LIN {X 0.032,Y -161.435,Z 1812.829,A 0.000,B 0.000,C 90.000,E1 149.282} C_DIS
LIN {X 0.039,Y -165.636,Z 1812.810,A 0.000,B 0.000,C 90.000,E1 145.754} C_DIS
LIN {X 0.022,Y -170.567,Z 1812.790,A 0.000,B 0.000,C 90.000,E1 142.271} C_DIS
LIN {X -0.071,Y -175.445,Z 1812.771,A 0.000,B 0.000,C 90.000,E1 138.852} C_DIS
LIN {X 0.045,Y -181.069,Z 1812.752,A 0.000,B 0.000,C 90.000,E1 135.405} C_DIS
LIN {X 0.036,Y -186.507,Z 1812.734,A 0.000,B 0.000,C 90.000,E1 132.043} C_DIS
LIN {X -0.021,Y -191.126,Z 1812.720,A 0.000,B 0.000,C 90.000,E1 129.564} C_DIS
LIN {X -0.101,Y -196.923,Z 1812.702,A 0.000,B 0.000,C 90.000,E1 126.297} C_DIS
LIN {X 0.093,Y -200.186,Z 1812.692,A 0.000,B 0.000,C 90.000,E1 124.612} C_DIS
LIN {X 0.089,Y -207.681,Z 1812.670,A 0.000,B 0.000,C 90.000,E1 120.590} C_DIS
LIN {X -0.010,Y -210.869,Z 1812.661,A 0.000,B 0.000,C 90.000,E1 119.027} C_DIS
LIN {X 0.101,Y -216.728,Z 1812.644,A 0.000,B 0.000,C 90.000,E1 115.848} C_DIS
LIN {X -0.080,Y -219.791,Z 1812.635,A 0.000,B 0.000,C 90.000,E1 114.335} C_DIS
LIN {X 0.010,Y -224.007,Z 1812.622,A 0.000,B 0.000,C 90.000,E1 111.897} C_DIS
LIN {X -0.023,Y -283.286,Z 1812.622,A 0.000,B 0.000,C 90.000,E1 111.897} C_DIS
LIN {X -0.096,Y -286.266,Z 1812.621,A 0.000,B 0.000,C 90.000,E1 111.844} C_DIS
LIN {X -0.059,Y -291.015,Z 1812.620,A 0.000,B 0.000,C 90.000,E1 111.535} C_DIS
LIN {X -0.019,Y -293.753,Z 1812.618,A 0.000,B 0.000,C 90.000,E1 111.227} C_DIS
LIN {X -0.009,Y -295.802,Z 1812.616,A 0.000,B 0.000,C 90.000,E1 110.918} C_DIS
LIN {X 0.132,Y -308.844,Z 1812.604,A 0.000,B 0.000,C 90.000,E1 108.598} C_DIS
LIN {X -0.084,Y -323.366,Z 1812.591,A 0.000,B 0.000,C 90.000,E1 106.370} C_DIS
LIN {X -0.136,Y -336.996,Z 1812.580,A 0.000,B 0.000,C 90.000,E1 104.481} C_DIS
LIN {X 0.084,Y -351.807,Z 1812.570,A 0.000,B 0.000,C 90.000,E1 102.591} C_DIS
LIN {X 0.058,Y -370.188,Z 1812.559,A 0.000,B 0.000,C 90.000,E1 100.546} C_DIS
LIN {X 0.090,Y -388.999,Z 1812.548,A 0.000,B 0.000,C 90.000,E1 98.681} C_DIS
LIN {X -0.052,Y -408.229,Z 1812.539,A 0.000,B 0.000,C 90.000,E1 97.004} C_DIS
LIN {X 0.143,Y -430.586,Z 1812.529,A 0.000,B 0.000,C 90.000,E1 95.220} C_DIS
LIN {X -0.141,Y -439.005,Z 1812.526,A 0.000,B 0.000,C 90.000,E1 94.645} C_DIS
LIN {X 0.070,Y -441.196,Z 1812.525,A 0.000,B 0.000,C 90.000,E1 94.416} C_DIS
LIN {X -0.017,Y -443.172,Z 1812.523,A 0.000,B 0.000,C 90.000,E1 94.188} C_DIS
LIN {X -0.073,Y -444.688,Z 1812.522,A 0.000,B 0.000,C 90.000,E1 93.955} C_DIS
LIN {X 0.104,Y -445.961,Z 1812.521,A 0.000,B 0.000,C 90.000,E1 93.669} C_DIS
LIN {X -0.162,Y -446.906,Z 1812.519,A 0.000,B 0.000,C 90.000,E1 93.440} C_DIS
LIN {X -0.206,Y -447.977,Z 1812.516,A 0.000,B 0.000,C 90.000,E1 92.922} C_DIS
LIN {X 0.178,Y -448.095,Z 1812.513,A 0.000,B 0.000,C 90.000,E1 92.350} C_DIS
LIN {X 0.126,Y -447.279,Z 1812.510,A 0.000,B 0.000,C 90.000,E1 91.835} C_DIS
LIN {X 0.086,Y -445.405,Z 1812.507,A 0.000,B 0.000,C 90.000,E1 91.318} C_DIS
LIN {X 0.029,Y -442.300,Z 1812.505,A 0.000,B 0.000,C 90.000,E1 90.802} C_DIS
LIN {X 0.055,Y -429.109,Z 1812.493,A 0.000,B 0.000,C 90.000,E1 88.682} C_DIS
LIN {X 0.115,Y -417.352,Z 1812.482,A 0.000,B 0.000,C 90.000,E1 86.788} C_DIS
LIN {X -0.123,Y -407.220,Z 1812.473,A 0.000,B 0.000,C 90.000,E1 85.179} C_DIS
LIN {X -0.062,Y -395.313,Z 1812.462,A 0.000,B 0.000,C 90.000,E1 83.223} C_DIS
LIN {X -0.160,Y -383.361,Z 1812.451,A 0.000,B 0.000,C 90.000,E1 81.254} C_DIS
LIN {X -0.061,Y -369.748,Z 1812.438,A 0.000,B 0.000,C 90.000,E1 78.926} C_DIS
LIN {X 0.062,Y -351.961,Z 1812.420,A 0.000,B 0.000,C 90.000,E1 75.644} C_DIS
LIN {X 0.049,Y -338.260,Z 1812.405,A 0.000,B 0.000,C 90.000,E1 72.906} C_DIS
LIN {X 0.047,Y -327.877,Z 1812.393,A 0.000,B 0.000,C 90.000,E1 70.732} C_DIS
LIN {X 0.147,Y -313.492,Z 1812.375,A 0.000,B 0.000,C 90.000,E1 67.539} C_DIS
LIN {X -0.191,Y -307.408,Z 1812.367,A 0.000,B 0.000,C 90.000,E1 66.177} C_DIS
LIN {X 0.160,Y -307.426,Z 1812.367,A 0.000,B 0.000,C 90.000,E1 66.102} C_DIS
LIN {X -0.061,Y -313.588,Z 1812.357,A 0.000,B 0.000,C 90.000,E1 64.332} C_DIS
LIN {X -0.097,Y -315.039,Z 1812.354,A 0.000,B 0.000,C 90.000,E1 63.691} C_DIS
LIN {X 0.156,Y -314.850,Z 1812.350,A 0.000,B 0.000,C 90.000,E1 62.999} C_DIS
LIN {X 0.136,Y -314.057,Z 1812.347,A 0.000,B 0.000,C 90.000,E1 62.359} C_DIS
LIN {X -0.163,Y -312.890,Z 1812.343,A 0.000,B 0.000,C 90.000,E1 61.769} C_DIS
LIN {X -0.040,Y -311.499,Z 1812.339,A 0.000,B 0.000,C 90.000,E1 61.101} C_DIS
LIN {X -0.077,Y -309.924,Z 1812.336,A 0.000,B 0.000,C 90.000,E1 60.461} C_DIS
LIN {X -0.029,Y -306.298,Z 1812.329,A 0.000,B 0.000,C 90.000,E1 59.154} C_DIS
LIN {X -0.131,Y -302.278,Z 1812.321,A 0.000,B 0.000,C 90.000,E1 57.867} C_DIS
LIN {X -0.082,Y -295.784,Z 1812.310,A 0.000,B 0.000,C 90.000,E1 55.881} C_DIS
LIN {X -0.007,Y -288.929,Z 1812.299,A 0.000,B 0.000,C 90.000,E1 53.863} C_DIS
LIN {X -0.008,Y -280.697,Z 1812.286,A 0.000,B 0.000,C 90.000,E1 51.492} C_DIS
LIN {X 0.037,Y -271.250,Z 1812.271,A 0.000,B 0.000,C 90.000,E1 48.728} C_DIS
LIN {X 0.001,Y -261.931,Z 1812.255,A 0.000,B 0.000,C 90.000,E1 45.931} C_DIS
LIN {X -0.082,Y -252.705,Z 1812.239,A 0.000,B 0.000,C 90.000,E1 43.095} C_DIS
LIN {X -0.014,Y -243.505,Z 1812.223,A 0.000,B 0.000,C 90.000,E1 40.172} C_DIS
LIN {X -0.137,Y -233.607,Z 1812.205,A 0.000,B 0.000,C 90.000,E1 36.870} C_DIS
LIN {X -0.042,Y -225.249,Z 1812.188,A 0.000,B 0.000,C 90.000,E1 33.833} C_DIS
LIN {X 0.033,Y -217.435,Z 1812.171,A 0.000,B 0.000,C 90.000,E1 30.747} C_DIS
LIN {X -0.006,Y -210.224,Z 1812.154,A 0.000,B 0.000,C 90.000,E1 27.641} C_DIS
LIN {X 0.043,Y -203.763,Z 1812.136,A 0.000,B 0.000,C 90.000,E1 24.463} C_DIS
LIN {X -0.047,Y -198.066,Z 1812.118,A 0.000,B 0.000,C 90.000,E1 21.280} C_DIS
LIN {X 0.062,Y -193.373,Z 1812.100,A 0.000,B 0.000,C 90.000,E1 18.000} C_DIS
LIN {X 0.064,Y -189.471,Z 1812.082,A 0.000,B 0.000,C 90.000,E1 14.717} C_DIS
LIN {X -0.020,Y -185.638,Z 1812.059,A 0.000,B 0.000,C 90.000,E1 10.602} C_DIS
LIN {X 0.045,Y -182.389,Z 1812.031,A 0.000,B 0.000,C 90.000,E1 5.568} C_DIS
LIN {X 0.015,Y -180.060,Z 1811.993,A 0.000,B 0.000,C 90.000,E1 358.682} C_DIS
LIN {X -0.031,Y -179.755,Z 1811.965,A 0.000,B 0.000,C 90.000,E1 353.628} C_DIS
LIN {X 0.009,Y -180.652,Z 1811.932,A 0.000,B 0.000,C 90.000,E1 347.701} C_DIS
LIN {X 0.001,Y -183.190,Z 1811.894,A 0.000,B 0.000,C 90.000,E1 340.967} C_DIS
LIN {X 0.075,Y -186.231,Z 1811.866,A 0.000,B 0.000,C 90.000,E1 335.921} C_DIS
LIN {X -0.051,Y -190.006,Z 1811.839,A 0.000,B 0.000,C 90.000,E1 330.973} C_DIS
LIN {X 0.006,Y -193.787,Z 1811.816,A 0.000,B 0.000,C 90.000,E1 326.834} C_DIS
LIN {X -0.044,Y -198.367,Z 1811.793,A 0.000,B 0.000,C 90.000,E1 322.763} C_DIS
LIN {X -0.102,Y -202.967,Z 1811.775,A 0.000,B 0.000,C 90.000,E1 319.542} C_DIS
LIN {X 0.000,Y -207.266,Z 1811.762,A 0.000,B 0.000,C 90.000,E1 317.106} C_DIS
LIN {X 0.102,Y -210.593,Z 1811.753,A 0.000,B 0.000,C 90.000,E1 315.486} C_DIS
LIN {X -0.006,Y -215.466,Z 1811.742,A 0.000,B 0.000,C 90.000,E1 313.542} C_DIS
LIN {X -0.087,Y -220.034,Z 1811.733,A 0.000,B 0.000,C 90.000,E1 312.000} C_DIS
LIN {X -0.108,Y -225.309,Z 1811.725,A 0.000,B 0.000,C 90.000,E1 310.458} C_DIS
LIN {X -0.036,Y -231.428,Z 1811.716,A 0.000,B 0.000,C 90.000,E1 308.910} C_DIS
LIN {X -0.060,Y -239.958,Z 1811.706,A 0.000,B 0.000,C 90.000,E1 307.030} C_DIS
LIN {X 0.061,Y -247.523,Z 1811.697,A 0.000,B 0.000,C 90.000,E1 305.518} C_DIS
LIN {X -0.111,Y -259.882,Z 1811.685,A 0.000,B 0.000,C 90.000,E1 303.372} C_DIS
LIN {X -0.111,Y -278.018,Z 1811.670,A 0.000,B 0.000,C 90.000,E1 300.541} C_DIS
LIN {X -0.137,Y -292.641,Z 1811.658,A 0.000,B 0.000,C 90.000,E1 298.487} C_DIS
LIN {X 0.030,Y -312.773,Z 1811.643,A 0.000,B 0.000,C 90.000,E1 295.796} C_DIS
LIN {X -0.102,Y -325.534,Z 1811.634,A 0.000,B 0.000,C 90.000,E1 294.207} C_DIS
LIN {X 0.124,Y -338.158,Z 1811.626,A 0.000,B 0.000,C 90.000,E1 292.589} C_DIS
LIN {X 0.124,Y -350.256,Z 1811.617,A 0.000,B 0.000,C 90.000,E1 291.046} C_DIS
LIN {X -0.127,Y -357.136,Z 1811.612,A 0.000,B 0.000,C 90.000,E1 290.174} C_DIS
LIN {X -0.100,Y -363.479,Z 1811.607,A 0.000,B 0.000,C 90.000,E1 289.268} C_DIS
LIN {X -0.016,Y -369.167,Z 1811.602,A 0.000,B 0.000,C 90.000,E1 288.362} C_DIS
LIN {X 0.133,Y -374.100,Z 1811.597,A 0.000,B 0.000,C 90.000,E1 287.457} C_DIS
LIN {X -0.141,Y -376.895,Z 1811.594,A 0.000,B 0.000,C 90.000,E1 286.913} C_DIS
LIN {X -0.035,Y -380.307,Z 1811.589,A 0.000,B 0.000,C 90.000,E1 286.024} C_DIS
LIN {X 0.093,Y -382.192,Z 1811.586,A 0.000,B 0.000,C 90.000,E1 285.426} C_DIS
LIN {X 0.227,Y -383.682,Z 1811.583,A 0.000,B 0.000,C 90.000,E1 284.828} C_DIS
LIN {X -0.099,Y -384.794,Z 1811.579,A 0.000,B 0.000,C 90.000,E1 284.300} C_DIS
LIN {X 0.053,Y -385.474,Z 1811.576,A 0.000,B 0.000,C 90.000,E1 283.703} C_DIS
LIN {X 0.119,Y -385.774,Z 1811.573,A 0.000,B 0.000,C 90.000,E1 283.119} C_DIS
LIN {X -0.184,Y -385.679,Z 1811.570,A 0.000,B 0.000,C 90.000,E1 282.591} C_DIS
LIN {X -0.109,Y -385.140,Z 1811.567,A 0.000,B 0.000,C 90.000,E1 282.007} C_DIS
LIN {X -0.032,Y -384.209,Z 1811.563,A 0.000,B 0.000,C 90.000,E1 281.422} C_DIS
LIN {X 0.040,Y -382.866,Z 1811.560,A 0.000,B 0.000,C 90.000,E1 280.838} C_DIS
LIN {X 0.106,Y -381.176,Z 1811.557,A 0.000,B 0.000,C 90.000,E1 280.254} C_DIS
LIN {X 0.183,Y -378.076,Z 1811.552,A 0.000,B 0.000,C 90.000,E1 279.378} C_DIS
LIN {X 0.168,Y -374.427,Z 1811.547,A 0.000,B 0.000,C 90.000,E1 278.511} C_DIS
LIN {X 0.118,Y -370.187,Z 1811.543,A 0.000,B 0.000,C 90.000,E1 277.644} C_DIS
LIN {X 0.037,Y -365.150,Z 1811.538,A 0.000,B 0.000,C 90.000,E1 276.777} C_DIS
LIN {X -0.093,Y -359.173,Z 1811.533,A 0.000,B 0.000,C 90.000,E1 275.910} C_DIS
LIN {X 0.136,Y -354.573,Z 1811.529,A 0.000,B 0.000,C 90.000,E1 275.277} C_DIS
LIN {X -0.016,Y -349.295,Z 1811.526,A 0.000,B 0.000,C 90.000,E1 274.702} C_DIS
LIN {X -0.063,Y -340.684,Z 1811.521,A 0.000,B 0.000,C 90.000,E1 273.841} C_DIS
LIN {X 0.124,Y -334.523,Z 1811.518,A 0.000,B 0.000,C 90.000,E1 273.269} C_DIS
LIN {X -0.040,Y -328.291,Z 1811.516,A 0.000,B 0.000,C 90.000,E1 272.808} C_DIS
LIN {X 0.015,Y -321.798,Z 1811.513,A 0.000,B 0.000,C 90.000,E1 272.350} C_DIS
LIN {X 0.017,Y -315.063,Z 1811.511,A 0.000,B 0.000,C 90.000,E1 271.949} C_DIS
LIN {X -0.002,Y -308.039,Z 1811.509,A 0.000,B 0.000,C 90.000,E1 271.604} C_DIS
LIN {X -0.036,Y -300.665,Z 1811.507,A 0.000,B 0.000,C 90.000,E1 271.318} C_DIS
LIN {X -0.024,Y -293.429,Z 1811.506,A 0.000,B 0.000,C 90.000,E1 271.088} C_DIS
LIN {X 0.084,Y -282.213,Z 1811.505,A 0.000,B 0.000,C 90.000,E1 270.802} C_DIS
LIN {X 0.083,Y -267.546,Z 1811.503,A 0.000,B 0.000,C 90.000,E1 270.516} C_DIS
LIN {X -0.067,Y -252.024,Z 1811.501,A 0.000,B 0.000,C 90.000,E1 270.286} C_DIS
LIN {X -0.055,Y -241.026,Z 1811.501,A 0.000,B 0.000,C 90.000,E1 270.172} C_DIS
LIN {X 0.028,Y -234.816,Z 1811.501,A 0.000,B 0.000,C 90.000,E1 270.115} C_DIS
LIN {X -0.002,Y -181.574,Z 1811.501,A 0.000,B 0.000,C 90.000,E1 270.115} C_DIS
LIN {X 0.084,Y -180.908,Z 1811.475,A 0.000,B 0.000,C 90.000,E1 265.527} C_DIS
LIN {X -0.038,Y -180.772,Z 1811.471,A 0.000,B 0.000,C 90.000,E1 264.723} C_DIS
LIN {X 0.033,Y -178.867,Z 1811.443,A 0.000,B 0.000,C 90.000,E1 259.634} C_DIS
LIN {X -0.066,Y -175.910,Z 1811.414,A 0.000,B 0.000,C 90.000,E1 254.574} C_DIS
LIN {X -0.010,Y -174.597,Z 1811.405,A 0.000,B 0.000,C 90.000,E1 252.851} C_DIS
LIN {X -0.083,Y -171.579,Z 1811.381,A 0.000,B 0.000,C 90.000,E1 248.592} C_DIS
LIN {X -0.093,Y -167.802,Z 1811.357,A 0.000,B 0.000,C 90.000,E1 244.280} C_DIS
LIN {X 0.072,Y -166.520,Z 1811.347,A 0.000,B 0.000,C 90.000,E1 242.487} C_DIS
LIN {X 0.060,Y -162.521,Z 1811.323,A 0.000,B 0.000,C 90.000,E1 238.122} C_DIS
LIN {X 0.031,Y -161.194,Z 1811.313,A 0.000,B 0.000,C 90.000,E1 236.373} C_DIS
LIN {X -0.066,Y -157.205,Z 1811.289,A 0.000,B 0.000,C 90.000,E1 231.984} C_DIS
LIN {X -0.043,Y -155.933,Z 1811.279,A 0.000,B 0.000,C 90.000,E1 230.194} C_DIS
LIN {X -0.083,Y -152.185,Z 1811.254,A 0.000,B 0.000,C 90.000,E1 225.729} C_DIS
LIN {X -0.062,Y -150.432,Z 1811.239,A 0.000,B 0.000,C 90.000,E1 223.014} C_DIS
LIN {X -0.033,Y -147.159,Z 1811.214,A 0.000,B 0.000,C 90.000,E1 218.463} C_DIS
LIN {X -0.067,Y -145.174,Z 1811.193,A 0.000,B 0.000,C 90.000,E1 214.818} C_DIS
LIN {X -0.031,Y -142.322,Z 1811.163,A 0.000,B 0.000,C 90.000,E1 209.283} C_DIS
LIN {X -0.037,Y -141.712,Z 1811.152,A 0.000,B 0.000,C 90.000,E1 207.436} C_DIS
LIN {X 0.012,Y -139.473,Z 1811.116,A 0.000,B 0.000,C 90.000,E1 200.918} C_DIS
LIN {X -0.067,Y -139.204,Z 1811.106,A 0.000,B 0.000,C 90.000,E1 199.087} C_DIS
LIN {X -0.008,Y -138.329,Z 1811.054,A 0.000,B 0.000,C 90.000,E1 189.726} C_DIS
LIN {X -0.005,Y -139.439,Z 1811.007,A 0.000,B 0.000,C 90.000,E1 181.318} C_DIS
LIN {X -0.066,Y -140.971,Z 1810.976,A 0.000,B 0.000,C 90.000,E1 175.755} C_DIS
LIN {X 0.025,Y -142.727,Z 1810.956,A 0.000,B 0.000,C 90.000,E1 172.008} C_DIS
LIN {X -0.017,Y -145.111,Z 1810.930,A 0.000,B 0.000,C 90.000,E1 167.409} C_DIS
LIN {X -0.022,Y -147.735,Z 1810.910,A 0.000,B 0.000,C 90.000,E1 163.740} C_DIS
LIN {X 0.059,Y -150.398,Z 1810.889,A 0.000,B 0.000,C 90.000,E1 160.061} C_DIS
LIN {X -0.066,Y -153.834,Z 1810.869,A 0.000,B 0.000,C 90.000,E1 156.485} C_DIS
LIN {X -0.007,Y -157.244,Z 1810.849,A 0.000,B 0.000,C 90.000,E1 152.871} C_DIS
LIN {X -0.067,Y -161.416,Z 1810.829,A 0.000,B 0.000,C 90.000,E1 149.331} C_DIS
LIN {X -0.057,Y -165.617,Z 1810.810,A 0.000,B 0.000,C 90.000,E1 145.801} C_DIS
LIN {X 0.063,Y -170.546,Z 1810.791,A 0.000,B 0.000,C 90.000,E1 142.271} C_DIS
LIN {X -0.029,Y -175.424,Z 1810.771,A 0.000,B 0.000,C 90.000,E1 138.852} C_DIS
LIN {X 0.088,Y -181.048,Z 1810.752,A 0.000,B 0.000,C 90.000,E1 135.405} C_DIS
LIN {X -0.046,Y -186.483,Z 1810.734,A 0.000,B 0.000,C 90.000,E1 132.081} C_DIS
LIN {X 0.022,Y -191.105,Z 1810.720,A 0.000,B 0.000,C 90.000,E1 129.564} C_DIS
LIN {X -0.057,Y -196.898,Z 1810.702,A 0.000,B 0.000,C 90.000,E1 126.297} C_DIS
LIN {X -0.026,Y -200.159,Z 1810.693,A 0.000,B 0.000,C 90.000,E1 124.659} C_DIS
LIN {X 0.030,Y -207.655,Z 1810.670,A 0.000,B 0.000,C 90.000,E1 120.620} C_DIS
LIN {X 0.037,Y -210.848,Z 1810.661,A 0.000,B 0.000,C 90.000,E1 119.027} C_DIS
LIN {X -0.047,Y -216.703,Z 1810.644,A 0.000,B 0.000,C 90.000,E1 115.899} C_DIS
LIN {X -0.033,Y -219.771,Z 1810.635,A 0.000,B 0.000,C 90.000,E1 114.335} C_DIS
LIN {X 0.002,Y -224.010,Z 1810.622,A 0.000,B 0.000,C 90.000,E1 111.897} C_DIS
LIN {X -0.033,Y -283.663,Z 1810.622,A 0.000,B 0.000,C 90.000,E1 111.897} C_DIS
LIN {X -0.036,Y -285.968,Z 1810.621,A 0.000,B 0.000,C 90.000,E1 111.844} C_DIS
LIN {X 0.003,Y -290.889,Z 1810.620,A 0.000,B 0.000,C 90.000,E1 111.535} C_DIS
LIN {X 0.044,Y -293.661,Z 1810.618,A 0.000,B 0.000,C 90.000,E1 111.227} C_DIS
LIN {X 0.069,Y -295.712,Z 1810.616,A 0.000,B 0.000,C 90.000,E1 110.918} C_DIS
LIN {X -0.065,Y -308.735,Z 1810.604,A 0.000,B 0.000,C 90.000,E1 108.652} C_DIS
LIN {X -0.076,Y -323.246,Z 1810.591,A 0.000,B 0.000,C 90.000,E1 106.386} C_DIS
LIN {X -0.037,Y -336.866,Z 1810.580,A 0.000,B 0.000,C 90.000,E1 104.481} C_DIS
LIN {X -0.158,Y -351.666,Z 1810.570,A 0.000,B 0.000,C 90.000,E1 102.647} C_DIS
LIN {X 0.155,Y -370.043,Z 1810.559,A 0.000,B 0.000,C 90.000,E1 100.546} C_DIS
LIN {X 0.125,Y -388.849,Z 1810.548,A 0.000,B 0.000,C 90.000,E1 98.690} C_DIS
LIN {X 0.037,Y -408.077,Z 1810.539,A 0.000,B 0.000,C 90.000,E1 97.004} C_DIS
LIN {X -0.200,Y -430.431,Z 1810.529,A 0.000,B 0.000,C 90.000,E1 95.277} C_DIS
LIN {X -0.057,Y -438.863,Z 1810.526,A 0.000,B 0.000,C 90.000,E1 94.645} C_DIS
LIN {X 0.153,Y -441.087,Z 1810.525,A 0.000,B 0.000,C 90.000,E1 94.416} C_DIS
LIN {X 0.084,Y -443.070,Z 1810.523,A 0.000,B 0.000,C 90.000,E1 94.188} C_DIS
LIN {X 0.047,Y -444.593,Z 1810.522,A 0.000,B 0.000,C 90.000,E1 93.955} C_DIS
LIN {X 0.224,Y -445.885,Z 1810.521,A 0.000,B 0.000,C 90.000,E1 93.669} C_DIS
LIN {X -0.042,Y -446.847,Z 1810.519,A 0.000,B 0.000,C 90.000,E1 93.440} C_DIS
LIN {X -0.087,Y -447.947,Z 1810.516,A 0.000,B 0.000,C 90.000,E1 92.922} C_DIS
LIN {X -0.150,Y -448.091,Z 1810.513,A 0.000,B 0.000,C 90.000,E1 92.407} C_DIS
LIN {X -0.203,Y -447.302,Z 1810.510,A 0.000,B 0.000,C 90.000,E1 91.892} C_DIS
LIN {X 0.204,Y -445.459,Z 1810.507,A 0.000,B 0.000,C 90.000,E1 91.318} C_DIS
LIN {X 0.147,Y -442.378,Z 1810.505,A 0.000,B 0.000,C 90.000,E1 90.802} C_DIS
LIN {X 0.172,Y -429.186,Z 1810.493,A 0.000,B 0.000,C 90.000,E1 88.682} C_DIS
LIN {X -0.187,Y -417.432,Z 1810.482,A 0.000,B 0.000,C 90.000,E1 86.846} C_DIS
LIN {X -0.010,Y -407.300,Z 1810.473,A 0.000,B 0.000,C 90.000,E1 85.179} C_DIS
LIN {X 0.050,Y -395.395,Z 1810.462,A 0.000,B 0.000,C 90.000,E1 83.223} C_DIS
LIN {X -0.050,Y -383.442,Z 1810.451,A 0.000,B 0.000,C 90.000,E1 81.254} C_DIS
LIN {X 0.047,Y -369.825,Z 1810.438,A 0.000,B 0.000,C 90.000,E1 78.926} C_DIS
LIN {X -0.174,Y -352.031,Z 1810.420,A 0.000,B 0.000,C 90.000,E1 75.700} C_DIS
LIN {X 0.152,Y -338.326,Z 1810.405,A 0.000,B 0.000,C 90.000,E1 72.906} C_DIS
LIN {X 0.148,Y -327.941,Z 1810.393,A 0.000,B 0.000,C 90.000,E1 70.732} C_DIS
LIN {X -0.098,Y -314.945,Z 1810.377,A 0.000,B 0.000,C 90.000,E1 67.922} C_DIS
LIN {X -0.035,Y -314.938,Z 1810.377,A 0.000,B 0.000,C 90.000,E1 67.901} C_DIS
LIN {X -0.040,Y -320.081,Z 1810.368,A 0.000,B 0.000,C 90.000,E1 66.305} C_DIS
LIN {X -0.040,Y -322.043,Z 1810.365,A 0.000,B 0.000,C 90.000,E1 65.665} C_DIS
LIN {X -0.029,Y -322.287,Z 1810.361,A 0.000,B 0.000,C 90.000,E1 65.025} C_DIS
LIN {X -0.143,Y -321.735,Z 1810.358,A 0.000,B 0.000,C 90.000,E1 64.409} C_DIS
LIN {X -0.119,Y -320.798,Z 1810.354,A 0.000,B 0.000,C 90.000,E1 63.768} C_DIS
LIN {X -0.097,Y -319.593,Z 1810.351,A 0.000,B 0.000,C 90.000,E1 63.127} C_DIS
LIN {X -0.074,Y -316.589,Z 1810.344,A 0.000,B 0.000,C 90.000,E1 61.847} C_DIS
LIN {X 0.058,Y -313.018,Z 1810.336,A 0.000,B 0.000,C 90.000,E1 60.539} C_DIS
LIN {X 0.034,Y -308.980,Z 1810.329,A 0.000,B 0.000,C 90.000,E1 59.253} C_DIS
LIN {X -0.151,Y -303.508,Z 1810.320,A 0.000,B 0.000,C 90.000,E1 57.661} C_DIS
LIN {X -0.095,Y -296.538,Z 1810.309,A 0.000,B 0.000,C 90.000,E1 55.674} C_DIS
LIN {X 0.157,Y -289.302,Z 1810.298,A 0.000,B 0.000,C 90.000,E1 53.623} C_DIS
LIN {X -0.053,Y -280.703,Z 1810.285,A 0.000,B 0.000,C 90.000,E1 51.295} C_DIS
LIN {X 0.006,Y -270.889,Z 1810.270,A 0.000,B 0.000,C 90.000,E1 48.528} C_DIS
LIN {X -0.031,Y -261.234,Z 1810.254,A 0.000,B 0.000,C 90.000,E1 45.729} C_DIS
LIN {X 0.049,Y -251.694,Z 1810.238,A 0.000,B 0.000,C 90.000,E1 42.852} C_DIS
LIN {X 0.076,Y -241.310,Z 1810.220,A 0.000,B 0.000,C 90.000,E1 39.564} C_DIS
LIN {X -0.047,Y -233.632,Z 1810.205,A 0.000,B 0.000,C 90.000,E1 36.996} C_DIS
LIN {X -0.085,Y -225.238,Z 1810.189,A 0.000,B 0.000,C 90.000,E1 33.992} C_DIS
LIN {X -0.077,Y -217.413,Z 1810.172,A 0.000,B 0.000,C 90.000,E1 30.924} C_DIS
LIN {X 0.066,Y -210.161,Z 1810.154,A 0.000,B 0.000,C 90.000,E1 27.769} C_DIS
LIN {X -0.074,Y -203.660,Z 1810.137,A 0.000,B 0.000,C 90.000,E1 24.643} C_DIS
LIN {X 0.019,Y -197.902,Z 1810.119,A 0.000,B 0.000,C 90.000,E1 21.408} C_DIS
LIN {X -0.059,Y -193.137,Z 1810.101,A 0.000,B 0.000,C 90.000,E1 18.181} C_DIS
LIN {X -0.059,Y -189.201,Z 1810.083,A 0.000,B 0.000,C 90.000,E1 14.898} C_DIS
LIN {X 0.037,Y -185.326,Z 1810.060,A 0.000,B 0.000,C 90.000,E1 10.725} C_DIS
LIN {X -0.062,Y -182.055,Z 1810.032,A 0.000,B 0.000,C 90.000,E1 5.739} C_DIS
LIN {X 0.013,Y -179.684,Z 1809.993,A 0.000,B 0.000,C 90.000,E1 358.682} C_DIS
LIN {X 0.018,Y -179.407,Z 1809.960,A 0.000,B 0.000,C 90.000,E1 352.761} C_DIS
LIN {X -0.022,Y -180.306,Z 1809.932,A 0.000,B 0.000,C 90.000,E1 347.701} C_DIS
LIN {X -0.050,Y -182.858,Z 1809.894,A 0.000,B 0.000,C 90.000,E1 340.967} C_DIS
LIN {X 0.011,Y -185.925,Z 1809.866,A 0.000,B 0.000,C 90.000,E1 335.921} C_DIS
LIN {X 0.039,Y -189.748,Z 1809.839,A 0.000,B 0.000,C 90.000,E1 330.923} C_DIS
LIN {X -0.080,Y -193.551,Z 1809.816,A 0.000,B 0.000,C 90.000,E1 326.834} C_DIS
LIN {X 0.019,Y -198.199,Z 1809.793,A 0.000,B 0.000,C 90.000,E1 322.718} C_DIS
LIN {X 0.084,Y -202.896,Z 1809.775,A 0.000,B 0.000,C 90.000,E1 319.461} C_DIS
LIN {X 0.039,Y -207.280,Z 1809.762,A 0.000,B 0.000,C 90.000,E1 317.067} C_DIS
LIN {X -0.003,Y -210.662,Z 1809.753,A 0.000,B 0.000,C 90.000,E1 315.486} C_DIS
LIN {X -0.109,Y -215.578,Z 1809.742,A 0.000,B 0.000,C 90.000,E1 313.542} C_DIS
LIN {X 0.124,Y -220.192,Z 1809.733,A 0.000,B 0.000,C 90.000,E1 311.919} C_DIS
LIN {X -0.038,Y -225.510,Z 1809.724,A 0.000,B 0.000,C 90.000,E1 310.415} C_DIS
LIN {X 0.007,Y -231.660,Z 1809.716,A 0.000,B 0.000,C 90.000,E1 308.874} C_DIS
LIN {X -0.017,Y -240.225,Z 1809.706,A 0.000,B 0.000,C 90.000,E1 306.996} C_DIS
LIN {X -0.043,Y -249.816,Z 1809.695,A 0.000,B 0.000,C 90.000,E1 305.152} C_DIS
LIN {X -0.071,Y -264.598,Z 1809.681,A 0.000,B 0.000,C 90.000,E1 302.625} C_DIS
LIN {X 0.059,Y -283.268,Z 1809.666,A 0.000,B 0.000,C 90.000,E1 299.795} C_DIS
LIN {X -0.003,Y -298.015,Z 1809.654,A 0.000,B 0.000,C 90.000,E1 297.769} C_DIS
LIN {X -0.015,Y -315.826,Z 1809.641,A 0.000,B 0.000,C 90.000,E1 295.463} C_DIS
LIN {X 0.186,Y -328.618,Z 1809.633,A 0.000,B 0.000,C 90.000,E1 293.823} C_DIS
LIN {X 0.052,Y -338.702,Z 1809.625,A 0.000,B 0.000,C 90.000,E1 292.589} C_DIS
LIN {X 0.058,Y -350.836,Z 1809.617,A 0.000,B 0.000,C 90.000,E1 291.046} C_DIS
LIN {X 0.146,Y -357.744,Z 1809.612,A 0.000,B 0.000,C 90.000,E1 290.120} C_DIS
LIN {X -0.158,Y -364.058,Z 1809.607,A 0.000,B 0.000,C 90.000,E1 289.268} C_DIS
LIN {X -0.068,Y -369.763,Z 1809.602,A 0.000,B 0.000,C 90.000,E1 288.362} C_DIS
LIN {X -0.012,Y -373.159,Z 1809.599,A 0.000,B 0.000,C 90.000,E1 287.764} C_DIS
LIN {X 0.174,Y -377.459,Z 1809.594,A 0.000,B 0.000,C 90.000,E1 286.858} C_DIS
LIN {X -0.076,Y -380.864,Z 1809.589,A 0.000,B 0.000,C 90.000,E1 286.024} C_DIS
LIN {X 0.056,Y -382.720,Z 1809.586,A 0.000,B 0.000,C 90.000,E1 285.426} C_DIS
LIN {X 0.193,Y -384.185,Z 1809.583,A 0.000,B 0.000,C 90.000,E1 284.828} C_DIS
LIN {X -0.129,Y -385.230,Z 1809.579,A 0.000,B 0.000,C 90.000,E1 284.300} C_DIS
LIN {X 0.026,Y -385.956,Z 1809.576,A 0.000,B 0.000,C 90.000,E1 283.703} C_DIS
LIN {X 0.095,Y -386.250,Z 1809.573,A 0.000,B 0.000,C 90.000,E1 283.119} C_DIS
LIN {X 0.171,Y -386.154,Z 1809.570,A 0.000,B 0.000,C 90.000,E1 282.535} C_DIS
LIN {X -0.127,Y -385.589,Z 1809.567,A 0.000,B 0.000,C 90.000,E1 282.007} C_DIS
LIN {X -0.049,Y -384.670,Z 1809.563,A 0.000,B 0.000,C 90.000,E1 281.422} C_DIS
LIN {X 0.026,Y -383.357,Z 1809.560,A 0.000,B 0.000,C 90.000,E1 280.838} C_DIS
LIN {X 0.095,Y -381.670,Z 1809.557,A 0.000,B 0.000,C 90.000,E1 280.254} C_DIS
LIN {X 0.154,Y -379.748,Z 1809.554,A 0.000,B 0.000,C 90.000,E1 279.670} C_DIS
LIN {X 0.154,Y -376.213,Z 1809.549,A 0.000,B 0.000,C 90.000,E1 278.803} C_DIS
LIN {X 0.125,Y -372.175,Z 1809.544,A 0.000,B 0.000,C 90.000,E1 277.936} C_DIS
LIN {X 0.058,Y -367.390,Z 1809.539,A 0.000,B 0.000,C 90.000,E1 277.068} C_DIS
LIN {X 0.020,Y -363.730,Z 1809.536,A 0.000,B 0.000,C 90.000,E1 276.486} C_DIS
LIN {X -0.154,Y -357.285,Z 1809.531,A 0.000,B 0.000,C 90.000,E1 275.625} C_DIS
LIN {X 0.067,Y -352.348,Z 1809.528,A 0.000,B 0.000,C 90.000,E1 274.992} C_DIS
LIN {X -0.090,Y -346.752,Z 1809.524,A 0.000,B 0.000,C 90.000,E1 274.416} C_DIS
LIN {X -0.020,Y -341.011,Z 1809.521,A 0.000,B 0.000,C 90.000,E1 273.841} C_DIS
LIN {X -0.125,Y -334.919,Z 1809.518,A 0.000,B 0.000,C 90.000,E1 273.326} C_DIS
LIN {X 0.059,Y -328.746,Z 1809.516,A 0.000,B 0.000,C 90.000,E1 272.808} C_DIS
LIN {X 0.100,Y -322.215,Z 1809.513,A 0.000,B 0.000,C 90.000,E1 272.350} C_DIS
LIN {X 0.104,Y -315.524,Z 1809.511,A 0.000,B 0.000,C 90.000,E1 271.949} C_DIS
LIN {X 0.069,Y -308.453,Z 1809.509,A 0.000,B 0.000,C 90.000,E1 271.604} C_DIS
LIN {X 0.003,Y -300.959,Z 1809.507,A 0.000,B 0.000,C 90.000,E1 271.318} C_DIS
LIN {X 0.009,Y -293.694,Z 1809.506,A 0.000,B 0.000,C 90.000,E1 271.088} C_DIS
LIN {X 0.012,Y -278.792,Z 1809.504,A 0.000,B 0.000,C 90.000,E1 270.745} C_DIS
LIN {X 0.003,Y -260.019,Z 1809.502,A 0.000,B 0.000,C 90.000,E1 270.401} C_DIS
LIN {X -0.049,Y -251.634,Z 1809.502,A 0.000,B 0.000,C 90.000,E1 270.286} C_DIS
LIN {X 0.096,Y -236.258,Z 1809.501,A 0.000,B 0.000,C 90.000,E1 270.115} C_DIS
LIN {X 0.066,Y -234.027,Z 1809.501,A 0.000,B 0.000,C 90.000,E1 270.115} C_DIS
LIN {X 0.028,Y -181.575,Z 1809.501,A 0.000,B 0.000,C 90.000,E1 270.115} C_DIS
LIN {X -0.065,Y -180.908,Z 1809.475,A 0.000,B 0.000,C 90.000,E1 265.584} C_DIS
LIN {X -0.008,Y -180.776,Z 1809.471,A 0.000,B 0.000,C 90.000,E1 264.723} C_DIS
LIN {X 0.063,Y -178.871,Z 1809.443,A 0.000,B 0.000,C 90.000,E1 259.634} C_DIS
LIN {X -0.035,Y -175.914,Z 1809.414,A 0.000,B 0.000,C 90.000,E1 254.574} C_DIS
LIN {X 0.021,Y -174.605,Z 1809.405,A 0.000,B 0.000,C 90.000,E1 252.851} C_DIS
LIN {X -0.053,Y -171.587,Z 1809.381,A 0.000,B 0.000,C 90.000,E1 248.592} C_DIS
LIN {X -0.064,Y -167.810,Z 1809.357,A 0.000,B 0.000,C 90.000,E1 244.280} C_DIS
LIN {X -0.047,Y -166.530,Z 1809.347,A 0.000,B 0.000,C 90.000,E1 242.538} C_DIS
LIN {X 0.090,Y -162.529,Z 1809.323,A 0.000,B 0.000,C 90.000,E1 238.122} C_DIS
LIN {X -0.074,Y -161.204,Z 1809.313,A 0.000,B 0.000,C 90.000,E1 236.421} C_DIS
LIN {X -0.038,Y -157.213,Z 1809.289,A 0.000,B 0.000,C 90.000,E1 231.984} C_DIS
LIN {X -0.015,Y -155.940,Z 1809.279,A 0.000,B 0.000,C 90.000,E1 230.194} C_DIS
LIN {X -0.055,Y -152.192,Z 1809.254,A 0.000,B 0.000,C 90.000,E1 225.729} C_DIS
LIN {X -0.034,Y -150.439,Z 1809.239,A 0.000,B 0.000,C 90.000,E1 223.014} C_DIS
LIN {X -0.006,Y -147.165,Z 1809.214,A 0.000,B 0.000,C 90.000,E1 218.463} C_DIS
LIN {X -0.040,Y -145.180,Z 1809.193,A 0.000,B 0.000,C 90.000,E1 214.818} C_DIS
LIN {X -0.005,Y -142.327,Z 1809.163,A 0.000,B 0.000,C 90.000,E1 209.283} C_DIS
LIN {X -0.009,Y -141.716,Z 1809.152,A 0.000,B 0.000,C 90.000,E1 207.436} C_DIS
LIN {X 0.038,Y -139.474,Z 1809.116,A 0.000,B 0.000,C 90.000,E1 200.918} C_DIS
LIN {X 0.029,Y -138.971,Z 1809.101,A 0.000,B 0.000,C 90.000,E1 198.127} C_DIS
LIN {X 0.018,Y -138.330,Z 1809.054,A 0.000,B 0.000,C 90.000,E1 189.726} C_DIS
LIN {X 0.021,Y -139.436,Z 1809.007,A 0.000,B 0.000,C 90.000,E1 181.318} C_DIS
LIN {X -0.039,Y -140.967,Z 1808.976,A 0.000,B 0.000,C 90.000,E1 175.755} C_DIS
LIN {X 0.052,Y -142.722,Z 1808.956,A 0.000,B 0.000,C 90.000,E1 172.008} C_DIS
LIN {X 0.010,Y -145.104,Z 1808.930,A 0.000,B 0.000,C 90.000,E1 167.409} C_DIS
LIN {X 0.005,Y -147.729,Z 1808.910,A 0.000,B 0.000,C 90.000,E1 163.740} C_DIS
LIN {X -0.054,Y -150.389,Z 1808.889,A 0.000,B 0.000,C 90.000,E1 160.115} C_DIS
LIN {X -0.038,Y -153.823,Z 1808.869,A 0.000,B 0.000,C 90.000,E1 156.485} C_DIS
LIN {X 0.021,Y -157.233,Z 1808.849,A 0.000,B 0.000,C 90.000,E1 152.871} C_DIS
LIN {X -0.038,Y -161.403,Z 1808.830,A 0.000,B 0.000,C 90.000,E1 149.331} C_DIS
LIN {X -0.028,Y -165.605,Z 1808.810,A 0.000,B 0.000,C 90.000,E1 145.801} C_DIS
LIN {X 0.093,Y -170.530,Z 1808.791,A 0.000,B 0.000,C 90.000,E1 142.271} C_DIS
LIN {X 0.001,Y -175.409,Z 1808.771,A 0.000,B 0.000,C 90.000,E1 138.852} C_DIS
LIN {X -0.009,Y -181.033,Z 1808.752,A 0.000,B 0.000,C 90.000,E1 135.445} C_DIS
LIN {X -0.014,Y -186.466,Z 1808.734,A 0.000,B 0.000,C 90.000,E1 132.081} C_DIS
LIN {X 0.054,Y -191.089,Z 1808.720,A 0.000,B 0.000,C 90.000,E1 129.564} C_DIS
LIN {X -0.025,Y -196.880,Z 1808.702,A 0.000,B 0.000,C 90.000,E1 126.297} C_DIS
LIN {X 0.007,Y -200.139,Z 1808.693,A 0.000,B 0.000,C 90.000,E1 124.659} C_DIS
LIN {X -0.116,Y -207.636,Z 1808.670,A 0.000,B 0.000,C 90.000,E1 120.669} C_DIS
LIN {X -0.114,Y -210.831,Z 1808.661,A 0.000,B 0.000,C 90.000,E1 119.077} C_DIS
LIN {X -0.013,Y -216.685,Z 1808.644,A 0.000,B 0.000,C 90.000,E1 115.899} C_DIS
LIN {X 0.003,Y -219.756,Z 1808.635,A 0.000,B 0.000,C 90.000,E1 114.335} C_DIS
LIN {X -0.035,Y -221.985,Z 1808.628,A 0.000,B 0.000,C 90.000,E1 113.025} C_DIS
LIN {X -0.081,Y -293.410,Z 1808.628,A 0.000,B 0.000,C 90.000,E1 113.025} C_DIS
LIN {X -0.036,Y -294.839,Z 1808.628,A 0.000,B 0.000,C 90.000,E1 113.003} C_DIS
LIN {X 0.082,Y -299.077,Z 1808.627,A 0.000,B 0.000,C 90.000,E1 112.770} C_DIS
LIN {X 0.086,Y -300.273,Z 1808.625,A 0.000,B 0.000,C 90.000,E1 112.461} C_DIS
LIN {X -0.153,Y -299.587,Z 1808.621,A 0.000,B 0.000,C 90.000,E1 111.844} C_DIS
LIN {X 0.092,Y -297.703,Z 1808.614,A 0.000,B 0.000,C 90.000,E1 110.556} C_DIS
LIN {X 0.039,Y -297.729,Z 1808.614,A 0.000,B 0.000,C 90.000,E1 110.556} C_DIS
LIN {X 0.100,Y -309.533,Z 1808.603,A 0.000,B 0.000,C 90.000,E1 108.489} C_DIS
LIN {X -0.093,Y -324.127,Z 1808.590,A 0.000,B 0.000,C 90.000,E1 106.260} C_DIS
LIN {X -0.042,Y -337.823,Z 1808.580,A 0.000,B 0.000,C 90.000,E1 104.356} C_DIS
LIN {X 0.116,Y -352.706,Z 1808.569,A 0.000,B 0.000,C 90.000,E1 102.479} C_DIS
LIN {X 0.155,Y -371.120,Z 1808.558,A 0.000,B 0.000,C 90.000,E1 100.433} C_DIS
LIN {X -0.128,Y -389.949,Z 1808.548,A 0.000,B 0.000,C 90.000,E1 98.624} C_DIS
LIN {X 0.183,Y -409.195,Z 1808.538,A 0.000,B 0.000,C 90.000,E1 96.891} C_DIS
LIN {X 0.024,Y -431.569,Z 1808.529,A 0.000,B 0.000,C 90.000,E1 95.163} C_DIS
LIN {X -0.020,Y -437.223,Z 1808.526,A 0.000,B 0.000,C 90.000,E1 94.759} C_DIS
LIN {X -0.024,Y -441.813,Z 1808.524,A 0.000,B 0.000,C 90.000,E1 94.359} C_DIS
LIN {X -0.044,Y -444.957,Z 1808.522,A 0.000,B 0.000,C 90.000,E1 93.898} C_DIS
LIN {X 0.131,Y -446.159,Z 1808.520,A 0.000,B 0.000,C 90.000,E1 93.612} C_DIS
LIN {X -0.140,Y -447.042,Z 1808.519,A 0.000,B 0.000,C 90.000,E1 93.383} C_DIS
LIN {X -0.183,Y -448.007,Z 1808.516,A 0.000,B 0.000,C 90.000,E1 92.865} C_DIS
LIN {X 0.204,Y -448.027,Z 1808.513,A 0.000,B 0.000,C 90.000,E1 92.293} C_DIS
LIN {X 0.164,Y -447.108,Z 1808.510,A 0.000,B 0.000,C 90.000,E1 91.776} C_DIS
LIN {X 0.110,Y -445.103,Z 1808.507,A 0.000,B 0.000,C 90.000,E1 91.260} C_DIS
LIN {X -0.023,Y -438.606,Z 1808.501,A 0.000,B 0.000,C 90.000,E1 90.229} C_DIS
LIN {X 0.207,Y -427.065,Z 1808.491,A 0.000,B 0.000,C 90.000,E1 88.339} C_DIS
LIN {X -0.191,Y -415.294,Z 1808.480,A 0.000,B 0.000,C 90.000,E1 86.502} C_DIS
LIN {X 0.036,Y -403.433,Z 1808.470,A 0.000,B 0.000,C 90.000,E1 84.546} C_DIS
LIN {X -0.007,Y -393.207,Z 1808.460,A 0.000,B 0.000,C 90.000,E1 82.875} C_DIS
LIN {X -0.141,Y -381.262,Z 1808.449,A 0.000,B 0.000,C 90.000,E1 80.905} C_DIS
LIN {X -0.106,Y -366.042,Z 1808.435,A 0.000,B 0.000,C 90.000,E1 78.285} C_DIS
LIN {X -0.023,Y -348.503,Z 1808.417,A 0.000,B 0.000,C 90.000,E1 74.991} C_DIS
LIN {X -0.014,Y -336.416,Z 1808.403,A 0.000,B 0.000,C 90.000,E1 72.543} C_DIS
LIN {X -0.091,Y -324.598,Z 1808.389,A 0.000,B 0.000,C 90.000,E1 70.061} C_DIS
LIN {X 0.028,Y -322.668,Z 1808.387,A 0.000,B 0.000,C 90.000,E1 69.625} C_DIS
LIN {X -0.027,Y -322.630,Z 1808.387,A 0.000,B 0.000,C 90.000,E1 69.625} C_DIS
LIN {X 0.134,Y -329.133,Z 1808.375,A 0.000,B 0.000,C 90.000,E1 67.486} C_DIS
LIN {X 0.053,Y -329.566,Z 1808.372,A 0.000,B 0.000,C 90.000,E1 66.869} C_DIS
LIN {X 0.115,Y -329.090,Z 1808.368,A 0.000,B 0.000,C 90.000,E1 66.230} C_DIS
LIN {X 0.049,Y -328.211,Z 1808.365,A 0.000,B 0.000,C 90.000,E1 65.613} C_DIS
LIN {X 0.114,Y -327.081,Z 1808.361,A 0.000,B 0.000,C 90.000,E1 64.973} C_DIS
LIN {X 0.088,Y -324.319,Z 1808.354,A 0.000,B 0.000,C 90.000,E1 63.717} C_DIS
LIN {X -0.117,Y -321.031,Z 1808.347,A 0.000,B 0.000,C 90.000,E1 62.487} C_DIS
LIN {X 0.076,Y -317.250,Z 1808.340,A 0.000,B 0.000,C 90.000,E1 61.179} C_DIS
LIN {X 0.015,Y -312.014,Z 1808.331,A 0.000,B 0.000,C 90.000,E1 59.587} C_DIS
LIN {X -0.134,Y -306.261,Z 1808.322,A 0.000,B 0.000,C 90.000,E1 57.995} C_DIS
LIN {X -0.030,Y -298.955,Z 1808.311,A 0.000,B 0.000,C 90.000,E1 56.008} C_DIS
LIN {X 0.098,Y -291.476,Z 1808.300,A 0.000,B 0.000,C 90.000,E1 53.989} C_DIS
LIN {X -0.071,Y -282.552,Z 1808.287,A 0.000,B 0.000,C 90.000,E1 51.662} C_DIS
LIN {X -0.147,Y -272.344,Z 1808.272,A 0.000,B 0.000,C 90.000,E1 48.933} C_DIS
LIN {X -0.148,Y -262.297,Z 1808.256,A 0.000,B 0.000,C 90.000,E1 46.134} C_DIS
LIN {X -0.025,Y -251.404,Z 1808.238,A 0.000,B 0.000,C 90.000,E1 42.894} C_DIS
LIN {X 0.019,Y -241.003,Z 1808.220,A 0.000,B 0.000,C 90.000,E1 39.600} C_DIS
LIN {X 0.033,Y -233.298,Z 1808.206,A 0.000,B 0.000,C 90.000,E1 36.996} C_DIS
LIN {X -0.015,Y -224.897,Z 1808.189,A 0.000,B 0.000,C 90.000,E1 33.992} C_DIS
LIN {X -0.018,Y -217.067,Z 1808.172,A 0.000,B 0.000,C 90.000,E1 30.924} C_DIS
LIN {X 0.115,Y -209.811,Z 1808.154,A 0.000,B 0.000,C 90.000,E1 27.769} C_DIS
LIN {X -0.034,Y -203.293,Z 1808.137,A 0.000,B 0.000,C 90.000,E1 24.643} C_DIS
LIN {X 0.047,Y -197.525,Z 1808.119,A 0.000,B 0.000,C 90.000,E1 21.408} C_DIS
LIN {X -0.040,Y -192.711,Z 1808.101,A 0.000,B 0.000,C 90.000,E1 18.181} C_DIS
LIN {X -0.050,Y -188.778,Z 1808.083,A 0.000,B 0.000,C 90.000,E1 14.898} C_DIS
LIN {X 0.033,Y -184.904,Z 1808.060,A 0.000,B 0.000,C 90.000,E1 10.725} C_DIS
LIN {X -0.081,Y -181.649,Z 1808.032,A 0.000,B 0.000,C 90.000,E1 5.739} C_DIS
LIN {X 0.010,Y -179.302,Z 1807.993,A 0.000,B 0.000,C 90.000,E1 358.682} C_DIS
LIN {X 0.063,Y -179.138,Z 1807.955,A 0.000,B 0.000,C 90.000,E1 351.894} C_DIS
LIN {X 0.043,Y -180.167,Z 1807.927,A 0.000,B 0.000,C 90.000,E1 346.825} C_DIS
LIN {X 0.074,Y -182.517,Z 1807.894,A 0.000,B 0.000,C 90.000,E1 340.913} C_DIS
LIN {X -0.052,Y -185.612,Z 1807.866,A 0.000,B 0.000,C 90.000,E1 335.921} C_DIS
LIN {X -0.037,Y -189.480,Z 1807.838,A 0.000,B 0.000,C 90.000,E1 330.923} C_DIS
LIN {X -0.003,Y -193.317,Z 1807.815,A 0.000,B 0.000,C 90.000,E1 326.786} C_DIS
LIN {X 0.044,Y -198.043,Z 1807.793,A 0.000,B 0.000,C 90.000,E1 322.683} C_DIS
LIN {X -0.017,Y -202.847,Z 1807.775,A 0.000,B 0.000,C 90.000,E1 319.461} C_DIS
LIN {X -0.066,Y -207.282,Z 1807.761,A 0.000,B 0.000,C 90.000,E1 317.067} C_DIS
LIN {X -0.041,Y -212.650,Z 1807.748,A 0.000,B 0.000,C 90.000,E1 314.676} C_DIS
LIN {X -0.010,Y -216.813,Z 1807.739,A 0.000,B 0.000,C 90.000,E1 313.095} C_DIS
LIN {X 0.078,Y -221.631,Z 1807.731,A 0.000,B 0.000,C 90.000,E1 311.515} C_DIS
LIN {X -0.070,Y -227.210,Z 1807.722,A 0.000,B 0.000,C 90.000,E1 310.011} C_DIS
LIN {X 0.029,Y -233.551,Z 1807.714,A 0.000,B 0.000,C 90.000,E1 308.463} C_DIS
LIN {X 0.045,Y -242.333,Z 1807.703,A 0.000,B 0.000,C 90.000,E1 306.583} C_DIS
LIN {X -0.081,Y -254.239,Z 1807.691,A 0.000,B 0.000,C 90.000,E1 304.405} C_DIS
LIN {X -0.002,Y -269.508,Z 1807.677,A 0.000,B 0.000,C 90.000,E1 301.878} C_DIS
LIN {X 0.121,Y -288.573,Z 1807.662,A 0.000,B 0.000,C 90.000,E1 299.077} C_DIS
LIN {X 0.044,Y -306.034,Z 1807.649,A 0.000,B 0.000,C 90.000,E1 296.744} C_DIS
LIN {X -0.201,Y -318.940,Z 1807.640,A 0.000,B 0.000,C 90.000,E1 295.155} C_DIS
LIN {X 0.052,Y -331.714,Z 1807.631,A 0.000,B 0.000,C 90.000,E1 293.515} C_DIS
LIN {X -0.051,Y -341.724,Z 1807.624,A 0.000,B 0.000,C 90.000,E1 292.280} C_DIS
LIN {X -0.008,Y -353.791,Z 1807.615,A 0.000,B 0.000,C 90.000,E1 290.737} C_DIS
LIN {X 0.114,Y -360.495,Z 1807.610,A 0.000,B 0.000,C 90.000,E1 289.812} C_DIS
LIN {X 0.171,Y -366.658,Z 1807.605,A 0.000,B 0.000,C 90.000,E1 288.906} C_DIS
LIN {X -0.144,Y -370.407,Z 1807.602,A 0.000,B 0.000,C 90.000,E1 288.362} C_DIS
LIN {X -0.085,Y -373.765,Z 1807.599,A 0.000,B 0.000,C 90.000,E1 287.764} C_DIS
LIN {X 0.106,Y -378.036,Z 1807.594,A 0.000,B 0.000,C 90.000,E1 286.858} C_DIS
LIN {X -0.139,Y -381.409,Z 1807.589,A 0.000,B 0.000,C 90.000,E1 286.024} C_DIS
LIN {X -0.004,Y -383.241,Z 1807.586,A 0.000,B 0.000,C 90.000,E1 285.426} C_DIS
LIN {X 0.137,Y -384.661,Z 1807.583,A 0.000,B 0.000,C 90.000,E1 284.828} C_DIS
LIN {X -0.182,Y -385.722,Z 1807.579,A 0.000,B 0.000,C 90.000,E1 284.300} C_DIS
LIN {X -0.026,Y -386.411,Z 1807.576,A 0.000,B 0.000,C 90.000,E1 283.703} C_DIS
LIN {X 0.047,Y -386.701,Z 1807.573,A 0.000,B 0.000,C 90.000,E1 283.119} C_DIS
LIN {X 0.125,Y -386.593,Z 1807.570,A 0.000,B 0.000,C 90.000,E1 282.535} C_DIS
LIN {X -0.170,Y -386.053,Z 1807.567,A 0.000,B 0.000,C 90.000,E1 282.007} C_DIS
LIN {X -0.088,Y -385.127,Z 1807.563,A 0.000,B 0.000,C 90.000,E1 281.422} C_DIS
LIN {X -0.010,Y -383.849,Z 1807.560,A 0.000,B 0.000,C 90.000,E1 280.838} C_DIS
LIN {X 0.061,Y -382.161,Z 1807.557,A 0.000,B 0.000,C 90.000,E1 280.254} C_DIS
LIN {X 0.149,Y -379.093,Z 1807.552,A 0.000,B 0.000,C 90.000,E1 279.378} C_DIS
LIN {X 0.143,Y -375.461,Z 1807.547,A 0.000,B 0.000,C 90.000,E1 278.511} C_DIS
LIN {X 0.102,Y -371.151,Z 1807.543,A 0.000,B 0.000,C 90.000,E1 277.644} C_DIS
LIN {X 0.030,Y -366.042,Z 1807.538,A 0.000,B 0.000,C 90.000,E1 276.777} C_DIS
LIN {X -0.057,Y -362.107,Z 1807.534,A 0.000,B 0.000,C 90.000,E1 276.201} C_DIS
LIN {X 0.142,Y -355.251,Z 1807.529,A 0.000,B 0.000,C 90.000,E1 275.277} C_DIS
LIN {X -0.002,Y -349.928,Z 1807.526,A 0.000,B 0.000,C 90.000,E1 274.702} C_DIS
LIN {X -0.057,Y -344.242,Z 1807.523,A 0.000,B 0.000,C 90.000,E1 274.131} C_DIS
LIN {X 0.126,Y -338.340,Z 1807.520,A 0.000,B 0.000,C 90.000,E1 273.555} C_DIS
LIN {X -0.143,Y -332.213,Z 1807.517,A 0.000,B 0.000,C 90.000,E1 273.094} C_DIS
LIN {X -0.147,Y -326.017,Z 1807.515,A 0.000,B 0.000,C 90.000,E1 272.636} C_DIS
LIN {X 0.090,Y -319.600,Z 1807.512,A 0.000,B 0.000,C 90.000,E1 272.178} C_DIS
LIN {X -0.077,Y -312.829,Z 1807.510,A 0.000,B 0.000,C 90.000,E1 271.835} C_DIS
LIN {X 0.037,Y -305.862,Z 1807.508,A 0.000,B 0.000,C 90.000,E1 271.489} C_DIS
LIN {X 0.141,Y -298.388,Z 1807.507,A 0.000,B 0.000,C 90.000,E1 271.203} C_DIS
LIN {X -0.067,Y -290.959,Z 1807.506,A 0.000,B 0.000,C 90.000,E1 271.031} C_DIS
LIN {X 0.051,Y -276.382,Z 1807.504,A 0.000,B 0.000,C 90.000,E1 270.688} C_DIS
LIN {X 0.108,Y -261.313,Z 1807.502,A 0.000,B 0.000,C 90.000,E1 270.401} C_DIS
LIN {X 0.035,Y -247.770,Z 1807.501,A 0.000,B 0.000,C 90.000,E1 270.229} C_DIS
LIN {X -0.114,Y -234.906,Z 1807.501,A 0.000,B 0.000,C 90.000,E1 270.172} C_DIS
LIN {X 0.090,Y -231.719,Z 1807.501,A 0.000,B 0.000,C 90.000,E1 270.115} C_DIS
LIN {X 0.046,Y -181.575,Z 1807.501,A 0.000,B 0.000,C 90.000,E1 270.115} C_DIS
LIN {X -0.024,Y -180.908,Z 1807.475,A 0.000,B 0.000,C 90.000,E1 265.584} C_DIS
LIN {X 0.034,Y -180.780,Z 1807.471,A 0.000,B 0.000,C 90.000,E1 264.723} C_DIS
LIN {X -0.071,Y -178.877,Z 1807.443,A 0.000,B 0.000,C 90.000,E1 259.690} C_DIS
LIN {X 0.005,Y -175.920,Z 1807.414,A 0.000,B 0.000,C 90.000,E1 254.574} C_DIS
LIN {X 0.061,Y -174.616,Z 1807.405,A 0.000,B 0.000,C 90.000,E1 252.851} C_DIS
LIN {X -0.014,Y -171.597,Z 1807.381,A 0.000,B 0.000,C 90.000,E1 248.592} C_DIS
LIN {X -0.024,Y -167.820,Z 1807.357,A 0.000,B 0.000,C 90.000,E1 244.280} C_DIS
LIN {X -0.007,Y -166.543,Z 1807.347,A 0.000,B 0.000,C 90.000,E1 242.538} C_DIS
LIN {X -0.096,Y -162.539,Z 1807.323,A 0.000,B 0.000,C 90.000,E1 238.201} C_DIS
LIN {X -0.036,Y -161.217,Z 1807.313,A 0.000,B 0.000,C 90.000,E1 236.421} C_DIS
LIN {X -0.001,Y -157.224,Z 1807.289,A 0.000,B 0.000,C 90.000,E1 231.984} C_DIS
LIN {X 0.023,Y -155.949,Z 1807.279,A 0.000,B 0.000,C 90.000,E1 230.194} C_DIS
LIN {X -0.018,Y -152.203,Z 1807.254,A 0.000,B 0.000,C 90.000,E1 225.729} C_DIS
LIN {X 0.003,Y -150.448,Z 1807.239,A 0.000,B 0.000,C 90.000,E1 223.014} C_DIS
LIN {X 0.029,Y -147.173,Z 1807.214,A 0.000,B 0.000,C 90.000,E1 218.463} C_DIS
LIN {X -0.004,Y -145.190,Z 1807.193,A 0.000,B 0.000,C 90.000,E1 214.818} C_DIS
LIN {X 0.031,Y -142.332,Z 1807.163,A 0.000,B 0.000,C 90.000,E1 209.283} C_DIS
LIN {X -0.039,Y -141.722,Z 1807.152,A 0.000,B 0.000,C 90.000,E1 207.462} C_DIS
LIN {X -0.057,Y -139.477,Z 1807.116,A 0.000,B 0.000,C 90.000,E1 200.972} C_DIS
LIN {X -0.068,Y -138.974,Z 1807.101,A 0.000,B 0.000,C 90.000,E1 198.181} C_DIS
LIN {X 0.053,Y -138.331,Z 1807.054,A 0.000,B 0.000,C 90.000,E1 189.726} C_DIS
LIN {X 0.056,Y -139.433,Z 1807.007,A 0.000,B 0.000,C 90.000,E1 181.318} C_DIS
LIN {X -0.003,Y -140.960,Z 1806.976,A 0.000,B 0.000,C 90.000,E1 175.755} C_DIS
LIN {X -0.053,Y -142.716,Z 1806.956,A 0.000,B 0.000,C 90.000,E1 172.064} C_DIS
LIN {X 0.046,Y -145.095,Z 1806.930,A 0.000,B 0.000,C 90.000,E1 167.409} C_DIS
LIN {X 0.041,Y -147.719,Z 1806.910,A 0.000,B 0.000,C 90.000,E1 163.740} C_DIS
LIN {X -0.017,Y -150.378,Z 1806.890,A 0.000,B 0.000,C 90.000,E1 160.115} C_DIS
LIN {X 0.000,Y -153.807,Z 1806.869,A 0.000,B 0.000,C 90.000,E1 156.485} C_DIS
LIN {X 0.059,Y -157.220,Z 1806.849,A 0.000,B 0.000,C 90.000,E1 152.871} C_DIS
LIN {X 0.001,Y -161.385,Z 1806.830,A 0.000,B 0.000,C 90.000,E1 149.331} C_DIS
LIN {X 0.012,Y -165.587,Z 1806.810,A 0.000,B 0.000,C 90.000,E1 145.801} C_DIS
LIN {X -0.002,Y -170.509,Z 1806.791,A 0.000,B 0.000,C 90.000,E1 142.316} C_DIS
LIN {X 0.042,Y -175.390,Z 1806.771,A 0.000,B 0.000,C 90.000,E1 138.852} C_DIS
LIN {X -0.096,Y -181.013,Z 1806.753,A 0.000,B 0.000,C 90.000,E1 135.486} C_DIS
LIN {X 0.028,Y -186.443,Z 1806.734,A 0.000,B 0.000,C 90.000,E1 132.081} C_DIS
LIN {X 0.098,Y -191.068,Z 1806.720,A 0.000,B 0.000,C 90.000,E1 129.564} C_DIS
LIN {X 0.019,Y -196.855,Z 1806.702,A 0.000,B 0.000,C 90.000,E1 126.297} C_DIS
LIN {X -0.063,Y -200.113,Z 1806.693,A 0.000,B 0.000,C 90.000,E1 124.692} C_DIS
LIN {X -0.070,Y -207.611,Z 1806.670,A 0.000,B 0.000,C 90.000,E1 120.669} C_DIS
LIN {X -0.068,Y -210.811,Z 1806.661,A 0.000,B 0.000,C 90.000,E1 119.077} C_DIS
LIN {X -0.061,Y -216.660,Z 1806.644,A 0.000,B 0.000,C 90.000,E1 115.924} C_DIS
LIN {X 0.064,Y -219.853,Z 1806.635,A 0.000,B 0.000,C 90.000,E1 114.259} C_DIS
LIN {X -0.105,Y -220.011,Z 1806.634,A 0.000,B 0.000,C 90.000,E1 114.207} C_DIS
LIN {X 0.078,Y -308.680,Z 1806.634,A 0.000,B 0.000,C 90.000,E1 114.155} C_DIS
LIN {X 0.035,Y -310.457,Z 1806.634,A 0.000,B 0.000,C 90.000,E1 114.131} C_DIS
LIN {X 0.173,Y -313.988,Z 1806.633,A 0.000,B 0.000,C 90.000,E1 113.823} C_DIS
LIN {X 0.023,Y -314.487,Z 1806.631,A 0.000,B 0.000,C 90.000,E1 113.567} C_DIS
LIN {X 0.003,Y -312.358,Z 1806.624,A 0.000,B 0.000,C 90.000,E1 112.280} C_DIS
LIN {X -0.054,Y -307.252,Z 1806.605,A 0.000,B 0.000,C 90.000,E1 108.906} C_DIS
LIN {X -0.109,Y -307.263,Z 1806.605,A 0.000,B 0.000,C 90.000,E1 108.906} C_DIS
LIN {X 0.097,Y -320.597,Z 1806.593,A 0.000,B 0.000,C 90.000,E1 106.749} C_DIS
LIN {X 0.181,Y -333.987,Z 1806.583,A 0.000,B 0.000,C 90.000,E1 104.828} C_DIS
LIN {X -0.068,Y -348.538,Z 1806.572,A 0.000,B 0.000,C 90.000,E1 103.008} C_DIS
LIN {X 0.096,Y -364.137,Z 1806.562,A 0.000,B 0.000,C 90.000,E1 101.186} C_DIS
LIN {X 0.095,Y -382.844,Z 1806.552,A 0.000,B 0.000,C 90.000,E1 99.265} C_DIS
LIN {X 0.019,Y -401.917,Z 1806.542,A 0.000,B 0.000,C 90.000,E1 97.530} C_DIS
LIN {X -0.120,Y -424.159,Z 1806.532,A 0.000,B 0.000,C 90.000,E1 95.739} C_DIS
LIN {X -0.160,Y -438.276,Z 1806.526,A 0.000,B 0.000,C 90.000,E1 94.702} C_DIS
LIN {X -0.182,Y -442.450,Z 1806.524,A 0.000,B 0.000,C 90.000,E1 94.302} C_DIS
LIN {X 0.143,Y -444.169,Z 1806.522,A 0.000,B 0.000,C 90.000,E1 94.012} C_DIS
LIN {X -0.007,Y -445.490,Z 1806.521,A 0.000,B 0.000,C 90.000,E1 93.784} C_DIS
LIN {X -0.087,Y -447.311,Z 1806.518,A 0.000,B 0.000,C 90.000,E1 93.269} C_DIS
LIN {X -0.135,Y -448.074,Z 1806.515,A 0.000,B 0.000,C 90.000,E1 92.751} C_DIS
LIN {X -0.194,Y -447.901,Z 1806.512,A 0.000,B 0.000,C 90.000,E1 92.236} C_DIS
LIN {X 0.214,Y -446.774,Z 1806.509,A 0.000,B 0.000,C 90.000,E1 91.661} C_DIS
LIN {X -0.036,Y -445.803,Z 1806.508,A 0.000,B 0.000,C 90.000,E1 91.432} C_DIS
LIN {X 0.160,Y -444.503,Z 1806.506,A 0.000,B 0.000,C 90.000,E1 91.146} C_DIS
LIN {X -0.201,Y -431.325,Z 1806.495,A 0.000,B 0.000,C 90.000,E1 89.083} C_DIS
LIN {X 0.200,Y -421.309,Z 1806.486,A 0.000,B 0.000,C 90.000,E1 87.421} C_DIS
LIN {X 0.100,Y -409.500,Z 1806.475,A 0.000,B 0.000,C 90.000,E1 85.527} C_DIS
LIN {X -0.199,Y -397.608,Z 1806.464,A 0.000,B 0.000,C 90.000,E1 83.628} C_DIS
LIN {X 0.134,Y -385.655,Z 1806.453,A 0.000,B 0.000,C 90.000,E1 81.602} C_DIS
LIN {X -0.163,Y -373.702,Z 1806.442,A 0.000,B 0.000,C 90.000,E1 79.634} C_DIS
LIN {X 0.126,Y -357.218,Z 1806.426,A 0.000,B 0.000,C 90.000,E1 76.645} C_DIS
LIN {X 0.075,Y -341.768,Z 1806.409,A 0.000,B 0.000,C 90.000,E1 73.630} C_DIS
LIN {X -0.084,Y -330.529,Z 1806.396,A 0.000,B 0.000,C 90.000,E1 71.329} C_DIS
LIN {X 0.173,Y -330.521,Z 1806.396,A 0.000,B 0.000,C 90.000,E1 71.275} C_DIS
LIN {X 0.160,Y -336.439,Z 1806.385,A 0.000,B 0.000,C 90.000,E1 69.263} C_DIS
LIN {X 0.127,Y -336.987,Z 1806.381,A 0.000,B 0.000,C 90.000,E1 68.646} C_DIS
LIN {X 0.106,Y -336.501,Z 1806.378,A 0.000,B 0.000,C 90.000,E1 68.028} C_DIS
LIN {X 0.088,Y -335.590,Z 1806.375,A 0.000,B 0.000,C 90.000,E1 67.411} C_DIS
LIN {X 0.037,Y -333.113,Z 1806.368,A 0.000,B 0.000,C 90.000,E1 66.177} C_DIS
LIN {X 0.087,Y -330.141,Z 1806.361,A 0.000,B 0.000,C 90.000,E1 64.921} C_DIS
LIN {X -0.051,Y -326.796,Z 1806.354,A 0.000,B 0.000,C 90.000,E1 63.691} C_DIS
LIN {X 0.069,Y -323.111,Z 1806.347,A 0.000,B 0.000,C 90.000,E1 62.410} C_DIS
LIN {X -0.143,Y -319.011,Z 1806.340,A 0.000,B 0.000,C 90.000,E1 61.179} C_DIS
LIN {X 0.094,Y -313.442,Z 1806.331,A 0.000,B 0.000,C 90.000,E1 59.537} C_DIS
LIN {X 0.164,Y -306.142,Z 1806.320,A 0.000,B 0.000,C 90.000,E1 57.582} C_DIS
LIN {X 0.029,Y -297.197,Z 1806.307,A 0.000,B 0.000,C 90.000,E1 55.308} C_DIS
LIN {X -0.113,Y -289.331,Z 1806.296,A 0.000,B 0.000,C 90.000,E1 53.336} C_DIS
LIN {X -0.052,Y -281.394,Z 1806.285,A 0.000,B 0.000,C 90.000,E1 51.295} C_DIS
LIN {X 0.019,Y -270.837,Z 1806.270,A 0.000,B 0.000,C 90.000,E1 48.528} C_DIS
LIN {X 0.021,Y -259.358,Z 1806.252,A 0.000,B 0.000,C 90.000,E1 45.364} C_DIS
LIN {X 0.058,Y -248.596,Z 1806.234,A 0.000,B 0.000,C 90.000,E1 42.123} C_DIS
LIN {X 0.021,Y -238.305,Z 1806.216,A 0.000,B 0.000,C 90.000,E1 38.830} C_DIS
LIN {X -0.015,Y -228.581,Z 1806.197,A 0.000,B 0.000,C 90.000,E1 35.471} C_DIS
LIN {X 0.014,Y -220.436,Z 1806.180,A 0.000,B 0.000,C 90.000,E1 32.418} C_DIS
LIN {X -0.030,Y -212.876,Z 1806.163,A 0.000,B 0.000,C 90.000,E1 29.333} C_DIS
LIN {X -0.009,Y -205.993,Z 1806.145,A 0.000,B 0.000,C 90.000,E1 26.181} C_DIS
LIN {X 0.119,Y -199.827,Z 1806.128,A 0.000,B 0.000,C 90.000,E1 22.950} C_DIS
LIN {X -0.032,Y -194.542,Z 1806.110,A 0.000,B 0.000,C 90.000,E1 19.758} C_DIS
LIN {X 0.071,Y -191.146,Z 1806.096,A 0.000,B 0.000,C 90.000,E1 17.275} C_DIS
LIN {X -0.016,Y -186.630,Z 1806.073,A 0.000,B 0.000,C 90.000,E1 13.175} C_DIS
LIN {X 0.098,Y -183.221,Z 1806.050,A 0.000,B 0.000,C 90.000,E1 8.973} C_DIS
LIN {X 0.082,Y -180.098,Z 1806.017,A 0.000,B 0.000,C 90.000,E1 3.094} C_DIS
LIN {X -0.003,Y -178.601,Z 1805.974,A 0.000,B 0.000,C 90.000,E1 355.298} C_DIS
LIN {X 0.078,Y -179.199,Z 1805.941,A 0.000,B 0.000,C 90.000,E1 349.342} C_DIS
LIN {X 0.022,Y -181.348,Z 1805.903,A 0.000,B 0.000,C 90.000,E1 342.598} C_DIS
LIN {X 0.068,Y -184.162,Z 1805.875,A 0.000,B 0.000,C 90.000,E1 337.539} C_DIS
LIN {X 0.039,Y -187.815,Z 1805.848,A 0.000,B 0.000,C 90.000,E1 332.538} C_DIS
LIN {X 0.000,Y -191.451,Z 1805.824,A 0.000,B 0.000,C 90.000,E1 328.408} C_DIS
LIN {X 0.083,Y -195.831,Z 1805.802,A 0.000,B 0.000,C 90.000,E1 324.276} C_DIS
LIN {X 0.014,Y -201.474,Z 1805.779,A 0.000,B 0.000,C 90.000,E1 320.231} C_DIS
LIN {X -0.063,Y -205.734,Z 1805.766,A 0.000,B 0.000,C 90.000,E1 317.838} C_DIS
LIN {X 0.085,Y -210.828,Z 1805.752,A 0.000,B 0.000,C 90.000,E1 315.405} C_DIS
LIN {X -0.018,Y -215.832,Z 1805.741,A 0.000,B 0.000,C 90.000,E1 313.461} C_DIS
LIN {X -0.091,Y -220.537,Z 1805.733,A 0.000,B 0.000,C 90.000,E1 311.919} C_DIS
LIN {X 0.065,Y -225.975,Z 1805.724,A 0.000,B 0.000,C 90.000,E1 310.334} C_DIS
LIN {X 0.023,Y -230.523,Z 1805.718,A 0.000,B 0.000,C 90.000,E1 309.197} C_DIS
LIN {X -0.008,Y -238.956,Z 1805.707,A 0.000,B 0.000,C 90.000,E1 307.317} C_DIS
LIN {X 0.090,Y -248.446,Z 1805.697,A 0.000,B 0.000,C 90.000,E1 305.438} C_DIS
LIN {X 0.083,Y -265.347,Z 1805.681,A 0.000,B 0.000,C 90.000,E1 302.546} C_DIS
LIN {X 0.100,Y -284.103,Z 1805.665,A 0.000,B 0.000,C 90.000,E1 299.745} C_DIS
LIN {X 0.064,Y -301.428,Z 1805.652,A 0.000,B 0.000,C 90.000,E1 297.385} C_DIS
LIN {X 0.081,Y -316.850,Z 1805.641,A 0.000,B 0.000,C 90.000,E1 295.412} C_DIS
LIN {X 0.003,Y -329.731,Z 1805.632,A 0.000,B 0.000,C 90.000,E1 293.823} C_DIS
LIN {X -0.137,Y -342.292,Z 1805.624,A 0.000,B 0.000,C 90.000,E1 292.280} C_DIS
LIN {X -0.111,Y -352.013,Z 1805.617,A 0.000,B 0.000,C 90.000,E1 291.046} C_DIS
LIN {X -0.014,Y -358.925,Z 1805.612,A 0.000,B 0.000,C 90.000,E1 290.120} C_DIS
LIN {X 0.034,Y -365.251,Z 1805.607,A 0.000,B 0.000,C 90.000,E1 289.214} C_DIS
LIN {X 0.139,Y -370.980,Z 1805.602,A 0.000,B 0.000,C 90.000,E1 288.308} C_DIS
LIN {X -0.051,Y -375.871,Z 1805.597,A 0.000,B 0.000,C 90.000,E1 287.457} C_DIS
LIN {X 0.046,Y -378.585,Z 1805.594,A 0.000,B 0.000,C 90.000,E1 286.858} C_DIS
LIN {X -0.195,Y -381.923,Z 1805.589,A 0.000,B 0.000,C 90.000,E1 286.024} C_DIS
LIN {X -0.057,Y -383.725,Z 1805.586,A 0.000,B 0.000,C 90.000,E1 285.426} C_DIS
LIN {X 0.087,Y -385.179,Z 1805.582,A 0.000,B 0.000,C 90.000,E1 284.828} C_DIS
LIN {X 0.144,Y -386.187,Z 1805.579,A 0.000,B 0.000,C 90.000,E1 284.245} C_DIS
LIN {X -0.070,Y -386.868,Z 1805.576,A 0.000,B 0.000,C 90.000,E1 283.703} C_DIS
LIN {X 0.005,Y -387.131,Z 1805.573,A 0.000,B 0.000,C 90.000,E1 283.119} C_DIS
LIN {X 0.087,Y -387.036,Z 1805.570,A 0.000,B 0.000,C 90.000,E1 282.535} C_DIS
LIN {X -0.207,Y -386.514,Z 1805.567,A 0.000,B 0.000,C 90.000,E1 282.007} C_DIS
LIN {X -0.122,Y -385.594,Z 1805.563,A 0.000,B 0.000,C 90.000,E1 281.422} C_DIS
LIN {X -0.040,Y -384.305,Z 1805.560,A 0.000,B 0.000,C 90.000,E1 280.838} C_DIS
LIN {X 0.034,Y -382.625,Z 1805.557,A 0.000,B 0.000,C 90.000,E1 280.254} C_DIS
LIN {X 0.125,Y -379.585,Z 1805.552,A 0.000,B 0.000,C 90.000,E1 279.378} C_DIS
LIN {X 0.124,Y -375.957,Z 1805.547,A 0.000,B 0.000,C 90.000,E1 278.511} C_DIS
LIN {X 0.088,Y -371.638,Z 1805.543,A 0.000,B 0.000,C 90.000,E1 277.644} C_DIS
LIN {X 0.021,Y -366.458,Z 1805.538,A 0.000,B 0.000,C 90.000,E1 276.777} C_DIS
LIN {X -0.063,Y -362.510,Z 1805.534,A 0.000,B 0.000,C 90.000,E1 276.201} C_DIS
LIN {X -0.167,Y -358.001,Z 1805.531,A 0.000,B 0.000,C 90.000,E1 275.625} C_DIS
LIN {X 0.058,Y -352.975,Z 1805.528,A 0.000,B 0.000,C 90.000,E1 274.992} C_DIS
LIN {X -0.029,Y -347.430,Z 1805.525,A 0.000,B 0.000,C 90.000,E1 274.416} C_DIS
LIN {X 0.071,Y -341.680,Z 1805.521,A 0.000,B 0.000,C 90.000,E1 273.841} C_DIS
LIN {X -0.014,Y -335.591,Z 1805.518,A 0.000,B 0.000,C 90.000,E1 273.326} C_DIS
LIN {X -0.155,Y -329.405,Z 1805.516,A 0.000,B 0.000,C 90.000,E1 272.865} C_DIS
LIN {X -0.096,Y -322.936,Z 1805.513,A 0.000,B 0.000,C 90.000,E1 272.407} C_DIS
LIN {X -0.116,Y -316.083,Z 1805.511,A 0.000,B 0.000,C 90.000,E1 272.007} C_DIS
LIN {X -0.112,Y -309.150,Z 1805.509,A 0.000,B 0.000,C 90.000,E1 271.661} C_DIS
LIN {X -0.139,Y -301.974,Z 1805.507,A 0.000,B 0.000,C 90.000,E1 271.375} C_DIS
LIN {X 0.099,Y -294.272,Z 1805.506,A 0.000,B 0.000,C 90.000,E1 271.088} C_DIS
LIN {X 0.110,Y -279.817,Z 1805.504,A 0.000,B 0.000,C 90.000,E1 270.745} C_DIS
LIN {X 0.098,Y -261.024,Z 1805.502,A 0.000,B 0.000,C 90.000,E1 270.401} C_DIS
LIN {X 0.052,Y -252.414,Z 1805.502,A 0.000,B 0.000,C 90.000,E1 270.286} C_DIS
LIN {X -0.034,Y -237.476,Z 1805.501,A 0.000,B 0.000,C 90.000,E1 270.172} C_DIS
LIN {X -0.092,Y -232.608,Z 1805.501,A 0.000,B 0.000,C 90.000,E1 270.172} C_DIS
LIN {X 0.087,Y -181.577,Z 1805.501,A 0.000,B 0.000,C 90.000,E1 270.115} C_DIS
LIN {X 0.016,Y -180.908,Z 1805.475,A 0.000,B 0.000,C 90.000,E1 265.584} C_DIS
LIN {X 0.075,Y -180.785,Z 1805.471,A 0.000,B 0.000,C 90.000,E1 264.723} C_DIS
LIN {X -0.031,Y -178.883,Z 1805.443,A 0.000,B 0.000,C 90.000,E1 259.690} C_DIS
LIN {X 0.044,Y -175.925,Z 1805.414,A 0.000,B 0.000,C 90.000,E1 254.574} C_DIS
LIN {X -0.010,Y -175.364,Z 1805.410,A 0.000,B 0.000,C 90.000,E1 253.740} C_DIS
LIN {X 0.048,Y -172.142,Z 1805.386,A 0.000,B 0.000,C 90.000,E1 249.444} C_DIS
LIN {X 0.026,Y -171.606,Z 1805.381,A 0.000,B 0.000,C 90.000,E1 248.592} C_DIS
LIN {X 0.013,Y -167.829,Z 1805.357,A 0.000,B 0.000,C 90.000,E1 244.280} C_DIS
LIN {X 0.032,Y -166.555,Z 1805.348,A 0.000,B 0.000,C 90.000,E1 242.538} C_DIS
LIN {X -0.059,Y -162.550,Z 1805.323,A 0.000,B 0.000,C 90.000,E1 238.201} C_DIS
LIN {X 0.002,Y -161.228,Z 1805.313,A 0.000,B 0.000,C 90.000,E1 236.421} C_DIS
LIN {X 0.036,Y -157.234,Z 1805.289,A 0.000,B 0.000,C 90.000,E1 231.984} C_DIS
LIN {X 0.060,Y -155.958,Z 1805.279,A 0.000,B 0.000,C 90.000,E1 230.194} C_DIS
LIN {X 0.018,Y -152.212,Z 1805.254,A 0.000,B 0.000,C 90.000,E1 225.729} C_DIS
LIN {X 0.038,Y -150.457,Z 1805.239,A 0.000,B 0.000,C 90.000,E1 223.014} C_DIS
LIN {X 0.065,Y -147.182,Z 1805.214,A 0.000,B 0.000,C 90.000,E1 218.463} C_DIS
LIN {X 0.031,Y -145.199,Z 1805.193,A 0.000,B 0.000,C 90.000,E1 214.818} C_DIS
LIN {X -0.058,Y -142.338,Z 1805.163,A 0.000,B 0.000,C 90.000,E1 209.333} C_DIS
LIN {X -0.005,Y -141.726,Z 1805.153,A 0.000,B 0.000,C 90.000,E1 207.462} C_DIS
LIN {X -0.023,Y -139.479,Z 1805.116,A 0.000,B 0.000,C 90.000,E1 200.972} C_DIS
LIN {X -0.034,Y -138.978,Z 1805.101,A 0.000,B 0.000,C 90.000,E1 198.181} C_DIS
LIN {X -0.049,Y -138.332,Z 1805.054,A 0.000,B 0.000,C 90.000,E1 189.782} C_DIS
LIN {X -0.048,Y -139.430,Z 1805.008,A 0.000,B 0.000,C 90.000,E1 181.375} C_DIS
LIN {X 0.004,Y -141.357,Z 1804.971,A 0.000,B 0.000,C 90.000,E1 174.837} C_DIS
LIN {X -0.019,Y -142.711,Z 1804.956,A 0.000,B 0.000,C 90.000,E1 172.064} C_DIS
LIN {X -0.060,Y -145.086,Z 1804.930,A 0.000,B 0.000,C 90.000,E1 167.465} C_DIS
LIN {X -0.065,Y -147.711,Z 1804.910,A 0.000,B 0.000,C 90.000,E1 163.795} C_DIS
LIN {X 0.018,Y -150.366,Z 1804.890,A 0.000,B 0.000,C 90.000,E1 160.115} C_DIS
LIN {X 0.037,Y -153.793,Z 1804.869,A 0.000,B 0.000,C 90.000,E1 156.485} C_DIS
LIN {X -0.043,Y -157.205,Z 1804.849,A 0.000,B 0.000,C 90.000,E1 152.922} C_DIS
LIN {X 0.038,Y -161.368,Z 1804.830,A 0.000,B 0.000,C 90.000,E1 149.331} C_DIS
LIN {X 0.050,Y -165.570,Z 1804.810,A 0.000,B 0.000,C 90.000,E1 145.801} C_DIS
LIN {X -0.067,Y -170.489,Z 1804.791,A 0.000,B 0.000,C 90.000,E1 142.351} C_DIS
LIN {X 0.082,Y -175.370,Z 1804.772,A 0.000,B 0.000,C 90.000,E1 138.852} C_DIS
LIN {X -0.055,Y -180.994,Z 1804.753,A 0.000,B 0.000,C 90.000,E1 135.486} C_DIS
LIN {X 0.069,Y -186.421,Z 1804.734,A 0.000,B 0.000,C 90.000,E1 132.081} C_DIS
LIN {X 0.017,Y -191.048,Z 1804.720,A 0.000,B 0.000,C 90.000,E1 129.600} C_DIS
LIN {X 0.061,Y -196.832,Z 1804.702,A 0.000,B 0.000,C 90.000,E1 126.297} C_DIS
LIN {X -0.020,Y -200.088,Z 1804.693,A 0.000,B 0.000,C 90.000,E1 124.692} C_DIS
LIN {X -0.027,Y -207.587,Z 1804.670,A 0.000,B 0.000,C 90.000,E1 120.669} C_DIS
LIN {X -0.024,Y -210.790,Z 1804.661,A 0.000,B 0.000,C 90.000,E1 119.077} C_DIS
LIN {X -0.011,Y -217.154,Z 1804.643,A 0.000,B 0.000,C 90.000,E1 115.668} C_DIS
LIN {X 0.027,Y -217.818,Z 1804.641,A 0.000,B 0.000,C 90.000,E1 115.335} C_DIS
LIN {X 0.003,Y -322.497,Z 1804.641,A 0.000,B 0.000,C 90.000,E1 115.335} C_DIS
LIN {X -0.110,Y -324.794,Z 1804.641,A 0.000,B 0.000,C 90.000,E1 115.335} C_DIS
LIN {X -0.098,Y -328.078,Z 1804.640,A 0.000,B 0.000,C 90.000,E1 115.155} C_DIS
LIN {X -0.091,Y -329.018,Z 1804.638,A 0.000,B 0.000,C 90.000,E1 114.823} C_DIS
LIN {X -0.106,Y -326.715,Z 1804.631,A 0.000,B 0.000,C 90.000,E1 113.567} C_DIS
LIN {X 0.140,Y -319.379,Z 1804.606,A 0.000,B 0.000,C 90.000,E1 109.087} C_DIS
LIN {X -0.086,Y -317.063,Z 1804.596,A 0.000,B 0.000,C 90.000,E1 107.330} C_DIS
LIN {X 0.161,Y -317.063,Z 1804.596,A 0.000,B 0.000,C 90.000,E1 107.275} C_DIS
LIN {X -0.119,Y -330.908,Z 1804.585,A 0.000,B 0.000,C 90.000,E1 105.300} C_DIS
LIN {X -0.025,Y -345.192,Z 1804.574,A 0.000,B 0.000,C 90.000,E1 103.411} C_DIS
LIN {X -0.012,Y -360.627,Z 1804.564,A 0.000,B 0.000,C 90.000,E1 101.591} C_DIS
LIN {X 0.140,Y -379.214,Z 1804.553,A 0.000,B 0.000,C 90.000,E1 99.613} C_DIS
LIN {X -0.122,Y -398.251,Z 1804.544,A 0.000,B 0.000,C 90.000,E1 97.871} C_DIS
LIN {X -0.091,Y -420.422,Z 1804.533,A 0.000,B 0.000,C 90.000,E1 96.024} C_DIS
LIN {X -0.072,Y -437.313,Z 1804.526,A 0.000,B 0.000,C 90.000,E1 94.759} C_DIS
LIN {X -0.075,Y -441.857,Z 1804.524,A 0.000,B 0.000,C 90.000,E1 94.359} C_DIS
LIN {X -0.119,Y -444.989,Z 1804.522,A 0.000,B 0.000,C 90.000,E1 93.898} C_DIS
LIN {X 0.056,Y -446.175,Z 1804.520,A 0.000,B 0.000,C 90.000,E1 93.612} C_DIS
LIN {X -0.215,Y -447.046,Z 1804.519,A 0.000,B 0.000,C 90.000,E1 93.383} C_DIS
LIN {X 0.189,Y -447.990,Z 1804.516,A 0.000,B 0.000,C 90.000,E1 92.808} C_DIS
LIN {X 0.128,Y -447.990,Z 1804.513,A 0.000,B 0.000,C 90.000,E1 92.293} C_DIS
LIN {X 0.089,Y -447.050,Z 1804.510,A 0.000,B 0.000,C 90.000,E1 91.776} C_DIS
LIN {X 0.035,Y -445.019,Z 1804.507,A 0.000,B 0.000,C 90.000,E1 91.260} C_DIS
LIN {X 0.073,Y -436.851,Z 1804.500,A 0.000,B 0.000,C 90.000,E1 89.943} C_DIS
LIN {X 0.131,Y -426.965,Z 1804.491,A 0.000,B 0.000,C 90.000,E1 88.339} C_DIS
LIN {X 0.148,Y -415.193,Z 1804.480,A 0.000,B 0.000,C 90.000,E1 86.445} C_DIS
LIN {X -0.132,Y -405.039,Z 1804.471,A 0.000,B 0.000,C 90.000,E1 84.837} C_DIS
LIN {X -0.082,Y -393.105,Z 1804.460,A 0.000,B 0.000,C 90.000,E1 82.875} C_DIS
LIN {X 0.160,Y -381.159,Z 1804.449,A 0.000,B 0.000,C 90.000,E1 80.849} C_DIS
LIN {X 0.178,Y -365.940,Z 1804.435,A 0.000,B 0.000,C 90.000,E1 78.229} C_DIS
LIN {X -0.097,Y -348.403,Z 1804.417,A 0.000,B 0.000,C 90.000,E1 74.991} C_DIS
LIN {X 0.179,Y -338.557,Z 1804.406,A 0.000,B 0.000,C 90.000,E1 72.960} C_DIS
LIN {X 0.122,Y -338.525,Z 1804.405,A 0.000,B 0.000,C 90.000,E1 72.960} C_DIS
LIN {X 0.105,Y -343.179,Z 1804.396,A 0.000,B 0.000,C 90.000,E1 71.275} C_DIS
LIN {X -0.002,Y -344.512,Z 1804.393,A 0.000,B 0.000,C 90.000,E1 70.678} C_DIS
LIN {X 0.014,Y -344.331,Z 1804.389,A 0.000,B 0.000,C 90.000,E1 70.061} C_DIS
LIN {X 0.040,Y -343.554,Z 1804.386,A 0.000,B 0.000,C 90.000,E1 69.444} C_DIS
LIN {X -0.056,Y -342.462,Z 1804.382,A 0.000,B 0.000,C 90.000,E1 68.847} C_DIS
LIN {X -0.023,Y -339.719,Z 1804.376,A 0.000,B 0.000,C 90.000,E1 67.614} C_DIS
LIN {X 0.111,Y -336.540,Z 1804.369,A 0.000,B 0.000,C 90.000,E1 66.357} C_DIS
LIN {X -0.131,Y -331.308,Z 1804.358,A 0.000,B 0.000,C 90.000,E1 64.537} C_DIS
LIN {X 0.044,Y -327.525,Z 1804.351,A 0.000,B 0.000,C 90.000,E1 63.256} C_DIS
LIN {X -0.117,Y -323.451,Z 1804.344,A 0.000,B 0.000,C 90.000,E1 62.025} C_DIS
LIN {X 0.035,Y -317.853,Z 1804.336,A 0.000,B 0.000,C 90.000,E1 60.411} C_DIS
LIN {X 0.127,Y -311.777,Z 1804.327,A 0.000,B 0.000,C 90.000,E1 58.791} C_DIS
LIN {X 0.124,Y -305.343,Z 1804.318,A 0.000,B 0.000,C 90.000,E1 57.168} C_DIS
LIN {X -0.028,Y -296.015,Z 1804.305,A 0.000,B 0.000,C 90.000,E1 54.895} C_DIS
LIN {X -0.020,Y -287.836,Z 1804.294,A 0.000,B 0.000,C 90.000,E1 52.889} C_DIS
LIN {X -0.163,Y -279.595,Z 1804.282,A 0.000,B 0.000,C 90.000,E1 50.884} C_DIS
LIN {X -0.011,Y -266.200,Z 1804.263,A 0.000,B 0.000,C 90.000,E1 47.391} C_DIS
LIN {X -0.117,Y -253.810,Z 1804.244,A 0.000,B 0.000,C 90.000,E1 43.866} C_DIS
LIN {X -0.023,Y -244.424,Z 1804.227,A 0.000,B 0.000,C 90.000,E1 40.943} C_DIS
LIN {X 0.021,Y -234.311,Z 1804.209,A 0.000,B 0.000,C 90.000,E1 37.604} C_DIS
LIN {X 0.072,Y -224.766,Z 1804.190,A 0.000,B 0.000,C 90.000,E1 34.199} C_DIS
LIN {X 0.064,Y -216.874,Z 1804.173,A 0.000,B 0.000,C 90.000,E1 31.131} C_DIS
LIN {X 0.007,Y -209.557,Z 1804.156,A 0.000,B 0.000,C 90.000,E1 28.025} C_DIS
LIN {X 0.038,Y -202.963,Z 1804.138,A 0.000,B 0.000,C 90.000,E1 24.847} C_DIS
LIN {X -0.066,Y -197.153,Z 1804.120,A 0.000,B 0.000,C 90.000,E1 21.663} C_DIS
LIN {X 0.088,Y -192.175,Z 1804.102,A 0.000,B 0.000,C 90.000,E1 18.362} C_DIS
LIN {X 0.063,Y -188.220,Z 1804.084,A 0.000,B 0.000,C 90.000,E1 15.079} C_DIS
LIN {X -0.016,Y -184.265,Z 1804.061,A 0.000,B 0.000,C 90.000,E1 10.950} C_DIS
LIN {X 0.019,Y -180.935,Z 1804.033,A 0.000,B 0.000,C 90.000,E1 5.910} C_DIS
LIN {X 0.005,Y -178.539,Z 1803.993,A 0.000,B 0.000,C 90.000,E1 358.682} C_DIS
LIN {X 0.080,Y -178.542,Z 1803.950,A 0.000,B 0.000,C 90.000,E1 351.027} C_DIS
LIN {X 0.072,Y -179.987,Z 1803.917,A 0.000,B 0.000,C 90.000,E1 345.102} C_DIS
LIN {X 0.039,Y -182.787,Z 1803.885,A 0.000,B 0.000,C 90.000,E1 339.209} C_DIS
LIN {X -0.030,Y -186.197,Z 1803.857,A 0.000,B 0.000,C 90.000,E1 334.204} C_DIS
LIN {X -0.040,Y -189.673,Z 1803.833,A 0.000,B 0.000,C 90.000,E1 330.049} C_DIS
LIN {X -0.053,Y -193.784,Z 1803.811,A 0.000,B 0.000,C 90.000,E1 325.928} C_DIS
LIN {X 0.013,Y -197.794,Z 1803.792,A 0.000,B 0.000,C 90.000,E1 322.637} C_DIS
LIN {X 0.044,Y -201.415,Z 1803.779,A 0.000,B 0.000,C 90.000,E1 320.194} C_DIS
LIN {X -0.012,Y -205.742,Z 1803.766,A 0.000,B 0.000,C 90.000,E1 317.796} C_DIS
LIN {X -0.019,Y -210.892,Z 1803.752,A 0.000,B 0.000,C 90.000,E1 315.405} C_DIS
LIN {X 0.034,Y -215.952,Z 1803.741,A 0.000,B 0.000,C 90.000,E1 313.419} C_DIS
LIN {X 0.116,Y -220.710,Z 1803.733,A 0.000,B 0.000,C 90.000,E1 311.838} C_DIS
LIN {X -0.040,Y -226.195,Z 1803.724,A 0.000,B 0.000,C 90.000,E1 310.334} C_DIS
LIN {X -0.082,Y -230.758,Z 1803.718,A 0.000,B 0.000,C 90.000,E1 309.197} C_DIS
LIN {X 0.031,Y -239.222,Z 1803.707,A 0.000,B 0.000,C 90.000,E1 307.282} C_DIS
LIN {X -0.005,Y -246.756,Z 1803.699,A 0.000,B 0.000,C 90.000,E1 305.804} C_DIS
LIN {X 0.048,Y -261.325,Z 1803.685,A 0.000,B 0.000,C 90.000,E1 303.245} C_DIS
LIN {X -0.138,Y -279.708,Z 1803.669,A 0.000,B 0.000,C 90.000,E1 300.463} C_DIS
LIN {X 0.113,Y -296.848,Z 1803.656,A 0.000,B 0.000,C 90.000,E1 298.025} C_DIS
LIN {X 0.073,Y -314.787,Z 1803.643,A 0.000,B 0.000,C 90.000,E1 295.720} C_DIS
LIN {X -0.029,Y -327.699,Z 1803.634,A 0.000,B 0.000,C 90.000,E1 294.131} C_DIS
LIN {X -0.083,Y -340.381,Z 1803.625,A 0.000,B 0.000,C 90.000,E1 292.567} C_DIS
LIN {X -0.190,Y -352.605,Z 1803.617,A 0.000,B 0.000,C 90.000,E1 291.046} C_DIS
LIN {X -0.036,Y -361.694,Z 1803.610,A 0.000,B 0.000,C 90.000,E1 289.812} C_DIS
LIN {X 0.030,Y -367.833,Z 1803.605,A 0.000,B 0.000,C 90.000,E1 288.906} C_DIS
LIN {X 0.165,Y -373.323,Z 1803.600,A 0.000,B 0.000,C 90.000,E1 288.000} C_DIS
LIN {X -0.112,Y -376.442,Z 1803.597,A 0.000,B 0.000,C 90.000,E1 287.457} C_DIS
LIN {X -0.011,Y -380.353,Z 1803.592,A 0.000,B 0.000,C 90.000,E1 286.567} C_DIS
LIN {X 0.118,Y -382.477,Z 1803.589,A 0.000,B 0.000,C 90.000,E1 285.969} C_DIS
LIN {X -0.108,Y -384.217,Z 1803.586,A 0.000,B 0.000,C 90.000,E1 285.426} C_DIS
LIN {X 0.039,Y -385.606,Z 1803.582,A 0.000,B 0.000,C 90.000,E1 284.828} C_DIS
LIN {X 0.100,Y -386.649,Z 1803.579,A 0.000,B 0.000,C 90.000,E1 284.245} C_DIS
LIN {X -0.112,Y -387.329,Z 1803.576,A 0.000,B 0.000,C 90.000,E1 283.703} C_DIS
LIN {X -0.034,Y -387.578,Z 1803.573,A 0.000,B 0.000,C 90.000,E1 283.119} C_DIS
LIN {X 0.050,Y -387.470,Z 1803.570,A 0.000,B 0.000,C 90.000,E1 282.535} C_DIS
LIN {X 0.138,Y -386.950,Z 1803.567,A 0.000,B 0.000,C 90.000,E1 281.951} C_DIS
LIN {X -0.154,Y -386.054,Z 1803.563,A 0.000,B 0.000,C 90.000,E1 281.422} C_DIS
LIN {X -0.069,Y -384.765,Z 1803.560,A 0.000,B 0.000,C 90.000,E1 280.838} C_DIS
LIN {X 0.009,Y -383.120,Z 1803.557,A 0.000,B 0.000,C 90.000,E1 280.254} C_DIS
LIN {X 0.104,Y -380.074,Z 1803.552,A 0.000,B 0.000,C 90.000,E1 279.378} C_DIS
LIN {X 0.108,Y -376.429,Z 1803.547,A 0.000,B 0.000,C 90.000,E1 278.511} C_DIS
LIN {X 0.076,Y -372.065,Z 1803.542,A 0.000,B 0.000,C 90.000,E1 277.644} C_DIS
LIN {X 0.022,Y -368.731,Z 1803.539,A 0.000,B 0.000,C 90.000,E1 277.068} C_DIS
LIN {X -0.070,Y -362.901,Z 1803.534,A 0.000,B 0.000,C 90.000,E1 276.201} C_DIS
LIN {X -0.171,Y -358.347,Z 1803.531,A 0.000,B 0.000,C 90.000,E1 275.625} C_DIS
LIN {X 0.058,Y -353.312,Z 1803.528,A 0.000,B 0.000,C 90.000,E1 274.992} C_DIS
LIN {X -0.092,Y -347.633,Z 1803.524,A 0.000,B 0.000,C 90.000,E1 274.416} C_DIS
LIN {X -0.006,Y -341.788,Z 1803.521,A 0.000,B 0.000,C 90.000,E1 273.841} C_DIS
LIN {X -0.069,Y -335.703,Z 1803.518,A 0.000,B 0.000,C 90.000,E1 273.326} C_DIS
LIN {X 0.134,Y -329.516,Z 1803.516,A 0.000,B 0.000,C 90.000,E1 272.808} C_DIS
LIN {X -0.126,Y -323.032,Z 1803.513,A 0.000,B 0.000,C 90.000,E1 272.407} C_DIS
LIN {X -0.108,Y -316.267,Z 1803.511,A 0.000,B 0.000,C 90.000,E1 272.007} C_DIS
LIN {X -0.101,Y -309.369,Z 1803.509,A 0.000,B 0.000,C 90.000,E1 271.661} C_DIS
LIN {X -0.141,Y -302.087,Z 1803.507,A 0.000,B 0.000,C 90.000,E1 271.375} C_DIS
LIN {X 0.058,Y -293.940,Z 1803.506,A 0.000,B 0.000,C 90.000,E1 271.088} C_DIS
LIN {X 0.087,Y -279.563,Z 1803.504,A 0.000,B 0.000,C 90.000,E1 270.745} C_DIS
LIN {X 0.100,Y -260.892,Z 1803.502,A 0.000,B 0.000,C 90.000,E1 270.401} C_DIS
LIN {X 0.053,Y -251.875,Z 1803.502,A 0.000,B 0.000,C 90.000,E1 270.286} C_DIS
LIN {X 0.093,Y -240.427,Z 1803.501,A 0.000,B 0.000,C 90.000,E1 270.172} C_DIS
LIN {X -0.049,Y -233.068,Z 1803.501,A 0.000,B 0.000,C 90.000,E1 270.172} C_DIS
LIN {X -0.060,Y -181.578,Z 1803.501,A 0.000,B 0.000,C 90.000,E1 270.172} C_DIS
LIN {X -0.091,Y -180.787,Z 1803.471,A 0.000,B 0.000,C 90.000,E1 264.780} C_DIS
LIN {X -0.018,Y -178.884,Z 1803.443,A 0.000,B 0.000,C 90.000,E1 259.690} C_DIS
LIN {X 0.059,Y -175.927,Z 1803.414,A 0.000,B 0.000,C 90.000,E1 254.574} C_DIS
LIN {X 0.004,Y -175.369,Z 1803.410,A 0.000,B 0.000,C 90.000,E1 253.740} C_DIS
LIN {X 0.062,Y -172.146,Z 1803.386,A 0.000,B 0.000,C 90.000,E1 249.444} C_DIS
LIN {X 0.040,Y -171.610,Z 1803.381,A 0.000,B 0.000,C 90.000,E1 248.592} C_DIS
LIN {X 0.028,Y -167.833,Z 1803.357,A 0.000,B 0.000,C 90.000,E1 244.280} C_DIS
LIN {X 0.045,Y -166.559,Z 1803.348,A 0.000,B 0.000,C 90.000,E1 242.538} C_DIS
LIN {X -0.045,Y -162.553,Z 1803.323,A 0.000,B 0.000,C 90.000,E1 238.201} C_DIS
LIN {X 0.015,Y -161.232,Z 1803.313,A 0.000,B 0.000,C 90.000,E1 236.421} C_DIS
LIN {X 0.050,Y -157.238,Z 1803.289,A 0.000,B 0.000,C 90.000,E1 231.984} C_DIS
LIN {X -0.027,Y -155.961,Z 1803.279,A 0.000,B 0.000,C 90.000,E1 230.231} C_DIS
LIN {X 0.030,Y -152.215,Z 1803.254,A 0.000,B 0.000,C 90.000,E1 225.729} C_DIS
LIN {X 0.051,Y -150.459,Z 1803.239,A 0.000,B 0.000,C 90.000,E1 223.014} C_DIS
LIN {X 0.078,Y -147.185,Z 1803.214,A 0.000,B 0.000,C 90.000,E1 218.463} C_DIS
LIN {X 0.044,Y -145.203,Z 1803.193,A 0.000,B 0.000,C 90.000,E1 214.818} C_DIS
LIN {X -0.046,Y -142.339,Z 1803.163,A 0.000,B 0.000,C 90.000,E1 209.333} C_DIS
LIN {X 0.007,Y -141.728,Z 1803.153,A 0.000,B 0.000,C 90.000,E1 207.462} C_DIS
LIN {X -0.011,Y -139.481,Z 1803.116,A 0.000,B 0.000,C 90.000,E1 200.972} C_DIS
LIN {X -0.022,Y -138.980,Z 1803.101,A 0.000,B 0.000,C 90.000,E1 198.181} C_DIS
LIN {X -0.037,Y -138.332,Z 1803.054,A 0.000,B 0.000,C 90.000,E1 189.782} C_DIS
LIN {X -0.036,Y -139.428,Z 1803.008,A 0.000,B 0.000,C 90.000,E1 181.375} C_DIS
LIN {X 0.017,Y -141.355,Z 1802.971,A 0.000,B 0.000,C 90.000,E1 174.837} C_DIS
LIN {X -0.007,Y -142.709,Z 1802.956,A 0.000,B 0.000,C 90.000,E1 172.064} C_DIS
LIN {X -0.048,Y -145.083,Z 1802.930,A 0.000,B 0.000,C 90.000,E1 167.465} C_DIS
LIN {X -0.052,Y -147.708,Z 1802.910,A 0.000,B 0.000,C 90.000,E1 163.795} C_DIS
LIN {X 0.032,Y -150.362,Z 1802.890,A 0.000,B 0.000,C 90.000,E1 160.115} C_DIS
LIN {X 0.050,Y -153.788,Z 1802.870,A 0.000,B 0.000,C 90.000,E1 156.485} C_DIS
LIN {X -0.030,Y -157.200,Z 1802.849,A 0.000,B 0.000,C 90.000,E1 152.922} C_DIS
LIN {X 0.052,Y -161.361,Z 1802.830,A 0.000,B 0.000,C 90.000,E1 149.331} C_DIS
LIN {X 0.064,Y -165.564,Z 1802.810,A 0.000,B 0.000,C 90.000,E1 145.801} C_DIS
LIN {X -0.054,Y -170.481,Z 1802.791,A 0.000,B 0.000,C 90.000,E1 142.351} C_DIS
LIN {X 0.096,Y -175.363,Z 1802.772,A 0.000,B 0.000,C 90.000,E1 138.852} C_DIS
LIN {X -0.041,Y -180.987,Z 1802.753,A 0.000,B 0.000,C 90.000,E1 135.486} C_DIS
LIN {X -0.055,Y -186.412,Z 1802.734,A 0.000,B 0.000,C 90.000,E1 132.123} C_DIS
LIN {X -0.116,Y -191.040,Z 1802.720,A 0.000,B 0.000,C 90.000,E1 129.644} C_DIS
LIN {X 0.077,Y -196.823,Z 1802.702,A 0.000,B 0.000,C 90.000,E1 126.297} C_DIS
LIN {X -0.005,Y -200.078,Z 1802.693,A 0.000,B 0.000,C 90.000,E1 124.692} C_DIS
LIN {X -0.011,Y -207.577,Z 1802.670,A 0.000,B 0.000,C 90.000,E1 120.669} C_DIS
LIN {X -0.008,Y -210.783,Z 1802.661,A 0.000,B 0.000,C 90.000,E1 119.077} C_DIS
LIN {X -0.042,Y -215.180,Z 1802.648,A 0.000,B 0.000,C 90.000,E1 116.668} C_DIS
LIN {X 0.182,Y -337.834,Z 1802.648,A 0.000,B 0.000,C 90.000,E1 116.616} C_DIS
LIN {X 0.013,Y -341.921,Z 1802.646,A 0.000,B 0.000,C 90.000,E1 116.283} C_DIS
LIN {X -0.001,Y -342.766,Z 1802.644,A 0.000,B 0.000,C 90.000,E1 115.924} C_DIS
LIN {X 0.151,Y -342.531,Z 1802.641,A 0.000,B 0.000,C 90.000,E1 115.283} C_DIS
LIN {X 0.115,Y -335.189,Z 1802.620,A 0.000,B 0.000,C 90.000,E1 111.589} C_DIS
LIN {X 0.100,Y -328.724,Z 1802.596,A 0.000,B 0.000,C 90.000,E1 107.221} C_DIS
LIN {X -0.114,Y -327.110,Z 1802.588,A 0.000,B 0.000,C 90.000,E1 105.843} C_DIS
LIN {X -0.170,Y -327.106,Z 1802.588,A 0.000,B 0.000,C 90.000,E1 105.843} C_DIS
LIN {X 0.084,Y -342.173,Z 1802.577,A 0.000,B 0.000,C 90.000,E1 103.772} C_DIS
LIN {X 0.017,Y -357.396,Z 1802.566,A 0.000,B 0.000,C 90.000,E1 101.951} C_DIS
LIN {X 0.000,Y -375.941,Z 1802.555,A 0.000,B 0.000,C 90.000,E1 99.962} C_DIS
LIN {X -0.055,Y -394.874,Z 1802.545,A 0.000,B 0.000,C 90.000,E1 98.163} C_DIS
LIN {X 0.181,Y -416.979,Z 1802.535,A 0.000,B 0.000,C 90.000,E1 96.258} C_DIS
LIN {X 0.053,Y -439.378,Z 1802.526,A 0.000,B 0.000,C 90.000,E1 94.588} C_DIS
LIN {X -0.172,Y -441.457,Z 1802.524,A 0.000,B 0.000,C 90.000,E1 94.416} C_DIS
LIN {X 0.120,Y -443.408,Z 1802.523,A 0.000,B 0.000,C 90.000,E1 94.131} C_DIS
LIN {X 0.002,Y -444.898,Z 1802.522,A 0.000,B 0.000,C 90.000,E1 93.898} C_DIS
LIN {X 0.182,Y -446.102,Z 1802.520,A 0.000,B 0.000,C 90.000,E1 93.612} C_DIS
LIN {X -0.084,Y -446.988,Z 1802.519,A 0.000,B 0.000,C 90.000,E1 93.383} C_DIS
LIN {X -0.128,Y -447.963,Z 1802.516,A 0.000,B 0.000,C 90.000,E1 92.865} C_DIS
LIN {X -0.190,Y -447.990,Z 1802.513,A 0.000,B 0.000,C 90.000,E1 92.350} C_DIS
LIN {X 0.219,Y -447.080,Z 1802.510,A 0.000,B 0.000,C 90.000,E1 91.776} C_DIS
LIN {X 0.164,Y -445.087,Z 1802.507,A 0.000,B 0.000,C 90.000,E1 91.260} C_DIS
LIN {X 0.030,Y -438.596,Z 1802.501,A 0.000,B 0.000,C 90.000,E1 90.229} C_DIS
LIN {X -0.169,Y -427.052,Z 1802.491,A 0.000,B 0.000,C 90.000,E1 88.396} C_DIS
LIN {X -0.142,Y -415.282,Z 1802.480,A 0.000,B 0.000,C 90.000,E1 86.502} C_DIS
LIN {X -0.009,Y -405.127,Z 1802.471,A 0.000,B 0.000,C 90.000,E1 84.837} C_DIS
LIN {X 0.039,Y -393.195,Z 1802.460,A 0.000,B 0.000,C 90.000,E1 82.875} C_DIS
LIN {X -0.097,Y -381.249,Z 1802.449,A 0.000,B 0.000,C 90.000,E1 80.905} C_DIS
LIN {X -0.062,Y -366.024,Z 1802.435,A 0.000,B 0.000,C 90.000,E1 78.285} C_DIS
LIN {X 0.017,Y -348.479,Z 1802.417,A 0.000,B 0.000,C 90.000,E1 74.991} C_DIS
LIN {X 0.083,Y -346.707,Z 1802.415,A 0.000,B 0.000,C 90.000,E1 74.629} C_DIS
LIN {X 0.026,Y -346.698,Z 1802.415,A 0.000,B 0.000,C 90.000,E1 74.629} C_DIS
LIN {X 0.097,Y -352.081,Z 1802.403,A 0.000,B 0.000,C 90.000,E1 72.543} C_DIS
LIN {X 0.045,Y -352.224,Z 1802.400,A 0.000,B 0.000,C 90.000,E1 71.945} C_DIS
LIN {X 0.113,Y -351.528,Z 1802.396,A 0.000,B 0.000,C 90.000,E1 71.329} C_DIS
LIN {X 0.071,Y -350.452,Z 1802.393,A 0.000,B 0.000,C 90.000,E1 70.732} C_DIS
LIN {X 0.082,Y -347.692,Z 1802.386,A 0.000,B 0.000,C 90.000,E1 69.518} C_DIS
LIN {X 0.183,Y -344.492,Z 1802.380,A 0.000,B 0.000,C 90.000,E1 68.284} C_DIS
LIN {X -0.053,Y -339.136,Z 1802.369,A 0.000,B 0.000,C 90.000,E1 66.485} C_DIS
LIN {X 0.053,Y -333.426,Z 1802.359,A 0.000,B 0.000,C 90.000,E1 64.613} C_DIS
LIN {X 0.039,Y -327.325,Z 1802.349,A 0.000,B 0.000,C 90.000,E1 62.743} C_DIS
LIN {X -0.030,Y -321.756,Z 1802.340,A 0.000,B 0.000,C 90.000,E1 61.179} C_DIS
LIN {X -0.034,Y -315.668,Z 1802.331,A 0.000,B 0.000,C 90.000,E1 59.587} C_DIS
LIN {X -0.081,Y -307.797,Z 1802.320,A 0.000,B 0.000,C 90.000,E1 57.661} C_DIS
LIN {X 0.046,Y -299.554,Z 1802.309,A 0.000,B 0.000,C 90.000,E1 55.674} C_DIS
LIN {X -0.059,Y -291.189,Z 1802.298,A 0.000,B 0.000,C 90.000,E1 53.703} C_DIS
LIN {X -0.015,Y -281.251,Z 1802.285,A 0.000,B 0.000,C 90.000,E1 51.331} C_DIS
LIN {X -0.077,Y -268.973,Z 1802.268,A 0.000,B 0.000,C 90.000,E1 48.243} C_DIS
LIN {X 0.087,Y -256.364,Z 1802.248,A 0.000,B 0.000,C 90.000,E1 44.676} C_DIS
LIN {X -0.129,Y -246.854,Z 1802.232,A 0.000,B 0.000,C 90.000,E1 41.838} C_DIS
LIN {X -0.031,Y -237.693,Z 1802.216,A 0.000,B 0.000,C 90.000,E1 38.874} C_DIS
END
